	10:	// Nowa operacja rozpoczęta - oczekiwanie na wkręcenie I śruby
		IF bScrewPass THEN
			I_PimSystem.mSetNewMachineState(nPIM_MachineStates._4_OperationInProgress);
			stFastenPIM_Data.i1ScrewPulses := iPassPulses;
			iWorkStep := 15;
		ELSIF NOT fbMotorSensorFilter.Q THEN
			mNewEvent(nEventClass:= nPIM_EventClasses.Error, nEvent:= nHIOS_ErrorList.MotorPulledFromFixWhenLocked);
		END_IF
	
	15:	// wkręcenie 2-giej śruby
		IF bScrewPass THEN
			stFastenPIM_Data.i2ScrewPulses := iPassPulses;
			iWorkStep := 20;
		ELSIF NOT fbMotorSensorFilter.Q THEN
			mNewEvent(nEventClass:= nPIM_EventClasses.Error, nEvent:= nHIOS_ErrorList.MotorPulledFromFixWhenLocked);
		END_IF
	
	20:	// Dwie śruby wkręcone prawidłowo
		I_PimSystem.mSetNewMachineState(nPIM_MachineStates._5_OperationEndedOK);
		iWorkStep := 30;

	30: // Zwolnienie części
		IF I_PimSystem.mSetNewMachineState(nPIM_MachineStates._6_ReturningToBaseState) THEN
			stDigInOuts.bMotorLockValve_Q := FALSE;	
			iWorkStep := 40;
		END_IF
				
	40:	// Operacja zakończona, status zapisany, idź do nowej operacji
		IF NOT fbMotorSensorFilter.Q THEN
			iWorkStep := 1;	
		END_IF	
		
	90:	//  blokowanie stanowiska
		stDigInOuts.bMotorLockValve_Q := TRUE;	
		fbTON_StepTimeout(IN:= FALSE);
		iTypZapytanie := 6;		// Zablokowanie wkrętaka
		iWorkStep := 91;
	
	91:	// Oczekiwanie na zapis statusu, wtedy wystawienie bitu blokowania
		IF I_PimSystem.mSetNewMachineState(nPIM_MachineStates._9_ResetInProgress) OR bServiceReset THEN
			fbTON_StepTimeout(IN:= FALSE);
			bServiceReset := FALSE;
			iWorkStep := 95;
		END_IF

	95:	// Potwierdzenie błędu
		fbTON_StepTimeout(IN:= TRUE, PT := T#2S);
		IF iTypZapytanie = 0 AND NOT bOczekiwanieNaOdpowiedz AND NOT bOdczytOK THEN
			iTypZapytanie := 7;		// Odblokowanie wkrętaka
		END_IF
		IF NOT bWkretakZablokowany THEN	
			stDigInOuts.bMotorLockValve_Q := FALSE;		
			
	
			nError := nHIOS_ErrorList.NoError;
			iWorkStep := 1;	
		END_IF
		IF fbTON_StepTimeout.Q THEN
			mNewEvent(nEventClass:= nPIM_EventClasses.Alarm, nEvent:= nHIOS_ErrorList.ResetTimeout);
		END_IF
		IF iWorkStep <> 95 THEN fbTON_StepTimeout(IN := FALSE); END_IF
	
	ELSE	// Krok domyślny w przypadku błędu w programie
		mNewEvent(nEventClass:= nPIM_EventClasses.Alarm, nEvent:= nHIOS_ErrorList.ProgramConfigError);
END_CASE

ACT_SerialCom();

// Zapis danych PIM	
IF bSqlExtDataSave THEN
	astExtData[1].sName := 'Hios-1Screw[Imp]';
	astExtData[1].sValue := INT_TO_STRING(stFastenPIM_Data.i1ScrewPulses);
	astExtData[2].sName := 'Hios-2Screw[Imp]';
	astExtData[2].sValue := INT_TO_STRING(stFastenPIM_Data.i2ScrewPulses);
	bSqlExtDataSavedOK := I_PimSystem.m_SqlInsertExtendedData(pParameters := ADR(astExtData), uiArraySize := SIZEOF(astExtData));
	bSqlExtDataSave := FALSE;
END_IF

IF GVL_Aircom.stAC_DT_Data.bNew_Shift THEN
	udiNbOfSavedOkStatusesMEM:= udiNbOfSavedOkStatuses;
	udiNbOfSavedNokStatusesMEM := udiNbOfSavedNokStatuses;
	udiNbOfSavedOkStatuses := udiNbOfSavedNokStatuses := 0;
END_IF

ACTION ACT_SerialCom:

IF bReadMachineParams THEN
	IF NOT bSendString AND NOT bOczekiwanieNaOdpowiedz AND NOT bWaitForAllParams THEN	// Start odczytu parametrów
		iTypZapytanie := 1;
		bWaitForAllParams := TRUE;
		iParamsCtr:= 0;
	END_IF
	fbTON_ParamsRead(IN:= bReadMachineParams, PT:= T#2S);
	IF bWaitForAllParams AND iParamsCtr >= 10 THEN			// Gdy wkrętak wysłał wszystkie parametry zakończ odczyt parametrów
		bReadMachineParams := bWaitForAllParams := FALSE;
		fbTON_ParamsRead(IN:=FALSE);
	END_IF
	IF fbTON_ParamsRead.Q THEN		// Parametry nie zostały odczytane
		bWaitForAllParams := bReadMachineParams := FALSE;
		fbTON_ParamsRead(IN:=FALSE);
	END_IF
END_IF

// Komunikacja *************************
fbRTRIG_NewSerialCmd(CLK:= iTypZapytanie <> 0);
bSendString S= fbRTRIG_NewSerialCmd.Q;
IF bSendString THEN
	CASE iTypZapytanie OF
		0:		// Bezczynność
		//	bSendString := FALSE;
		1:		// Zapytanie o parametry
			sSendingString := 'QS$N';
			MEMSET(destAddr := ADR(stScrewDriverParamsAct), fillByte := 0, n := SIZEOF(stScrewDriverParamsAct));
		2:		// Zapytanie o ilosc zalaczen wkretaka
			sSendingString := 'QL$N';
		3:		// Zapytanie o typ wkretaka
			sSendingString := 'QV$N';
		4:		// Reset bledu
			sSendingString := 'R:E$N';
		5:		// Reset licznika śrub do wkręcenia
			sSendingString := 'R:C$N';
		6:		// Zablokowanie wkretaka
			sSendingString := 'Lv:1$N';
		7:		// Odblokowanie wkretaka
			sSendingString := 'Lv:0$N';		
	END_CASE
	
	IF NOT fbSendString.Busy THEN
		sSendStringfb:= sSendingString;
	END_IF
	fbSendString(
		SendString := sSendStringfb,
		TXbuffer := stDigInOuts.stSerialCom.TxBufferEL);
	IF NOT fbSendString.Busy AND (fbSendString.Error = ComError_t.COMERROR_NOERROR) THEN
		MEMMOVE(srcAddr := ADR(asComunicationHistoryOut[1]), destAddr := ADR(asComunicationHistoryOut[2]),n:= 9* SIZEOF(asComunicationHistoryOut[1]));
		asComunicationHistoryOut[1]:= sSendStringfb;
		bSendString := FALSE;
		bOczekiwanieNaOdpowiedz:=TRUE;	
	ELSIF NOT fbSendString.Busy AND (fbSendString.Error <> ComError_t.COMERROR_NOERROR) THEN
		bSendString := FALSE;
		iTypZapytanie := 0;
		fbRTRIG_NewSerialCmd(CLK := FALSE);
		bOczekiwanieNaOdpowiedz:=FALSE;
		iComSendError := fbSendString.Error;	
	END_IF
END_IF 

fbRecvString(Prefix :='',
		Suffix := '$N',
		Timeout := T#1S,
		Reset := ,
		StringReceived =>,
		Busy =>,
		RXbuffer := stDigInOuts.stSerialCom.RxBufferEL,
		ReceivedString := sRcvString);

// Sprawdzenie poprawności komunikacji oraz odebranych danych
fbTON_Timer_Comm(IN := bSendString OR bOczekiwanieNaOdpowiedz, PT:= T#2S);

IF fbTON_Timer_Comm.Q THEN
	bQBladKomunikacji := TRUE;
	bOczekiwanieNaOdpowiedz := FALSE;
	bSendString:= FALSE;
	bOdczytOK := FALSE;
	fbRTRIG_NewSerialCmd(CLK := FALSE);
	iTypZapytanie := 0;
END_IF
// Dekodowanie odebranych informacji
bTorqueUp := bScrewFail := bScrewPass := FALSE;
bOdczytOK := FALSE;
IF fbRecvString.StringReceived THEN
	sRcvString := DELETE(STR:= sRcvString, LEN:=1, POS:= LEN(sRcvString));
	MEMMOVE(srcAddr := ADR(asComunicationHistoryIn[1]), destAddr := ADR(asComunicationHistoryIn[2]),n:= 9* SIZEOF(asComunicationHistoryIn[1]));
	asComunicationHistoryIn[1]:= sRcvString;
	bQBladKomunikacji := FALSE;
	bOczekiwanieNaOdpowiedz := FALSE;
	bOdczytOK := TRUE;
	iTypZapytanie := 0;
	// Wyłuskanie parametrow
	// Actual values	
	IF FIND(sRcvString, 'Lv:') > 0 THEN			// Określenie czy wkretak jest zablokowany
		sStringToRead := DELETE(STR:= sRcvString, LEN := 3, POS :=1);
		bWkretakZablokowany := STRING_TO_INT(sStringToRead) > 0;
	ELSIF FIND(sRcvString, 'AL:') > 0 THEN		// Licznik uruchomień
		sStringToRead := DELETE(STR:= sRcvString, LEN := 3, POS :=1);
		diStartsUpCtr := STRING_TO_DINT(sStringToRead);	
	ELSIF FIND(sRcvString, 'L:') > 0 THEN			// Określenie czy wkretak jest wlaczony
		sStringToRead := DELETE(STR:= sRcvString, LEN := 2, POS :=1);
		IF STRING_TO_INT(sStringToRead) > 0 THEN
			bWkretakWlaczony := TRUE;
			diStartsUpCtr := diStartsUpCtr +1;
		ELSE
			bWkretakWlaczony := FALSE;
		END_IF
	ELSIF FIND(sRcvString, 'Pulse:') > 0 THEN			// Aktualny licznik impulsow
		sStringToRead := DELETE(STR:= sRcvString, LEN := 6, POS :=1);
		iActPulses:= STRING_TO_INT(sStringToRead);
	ELSIF FIND(sRcvString, 'PASS') > 0 THEN			// Śruba wkręcona prawidlowo
		bScrewPass := TRUE;
	ELSIF FIND(sRcvString, 'FAIL') > 0 THEN			// Śruba wkręcona błędnie
		bScrewFail := TRUE;
	ELSIF FIND(sRcvString, 'E:  ,') > 0 THEN		// Licznik impulsow - bledna sruba
		sStringToRead := DELETE(STR:= sRcvString, LEN := 5, POS :=1);
		iFailPulses:= STRING_TO_INT(sStringToRead);
	ELSIF FIND(sRcvString, 'D:') > 0 THEN		// Licznik impulsow - dobra sruba
		sStringToRead := DELETE(STR:= sRcvString, LEN := 7, POS :=1);
		iPassPulses:= STRING_TO_INT(sStringToRead);
	ELSIF FIND(sRcvString, 'T') > 0 THEN		// Osiagnieto moment
		bTorqueUp:= TRUE;
	// Parameters
	ELSIF FIND(sRcvString, 'AR:') > 0 THEN			// Maksymalna liczba impulsow
		sStringToRead := DELETE(STR:= sRcvString, LEN := 3, POS :=1);
		stScrewDriverParamsAct.iSystemConstAR := STRING_TO_INT(sStringToRead);
		iParamsCtr := iParamsCtr + 1;
	ELSIF FIND(sRcvString, 'An:') > 0 THEN			// Liczba śrub do wkrecenia
		sStringToRead := DELETE(STR:= sRcvString, LEN := 3, POS :=1);
		stScrewDriverParamsAct.iScrewsToFastenAn := STRING_TO_INT(sStringToRead);
		iParamsCtr := iParamsCtr + 1;
	ELSIF FIND(sRcvString, 'Ac:') > 0 THEN			// Minimalna liczba impulsow
		sStringToRead := DELETE(STR:= sRcvString, LEN := 3, POS :=1);
		stScrewDriverParamsAct.iMinPulseAc := STRING_TO_INT(sStringToRead);
		iParamsCtr := iParamsCtr + 1;
	ELSIF FIND(sRcvString, 'AC:') > 0 THEN			// Maksymalna liczba impulsow
		sStringToRead := DELETE(STR:= sRcvString, LEN := 3, POS :=1);
		stScrewDriverParamsAct.iMaxPulseAC := STRING_TO_INT(sStringToRead);
		iParamsCtr := iParamsCtr + 1;
	ELSIF FIND(sRcvString, 'At:') > 0 THEN			// Work reset time
		sStringToRead := DELETE(STR:= sRcvString, LEN := 3, POS :=1);
		stScrewDriverParamsAct.iBuzzerScrewsDoneTimeAt := STRING_TO_INT(sStringToRead);
		iParamsCtr := iParamsCtr + 1;
	ELSIF FIND(sRcvString, 'Ar:') > 0 THEN			// Count time for reverse operation
		sStringToRead := DELETE(STR:= sRcvString, LEN := 3, POS :=1);
		stScrewDriverParamsAct.iCntTimeForReverseOperationAr := STRING_TO_INT(sStringToRead);
		iParamsCtr := iParamsCtr + 1;
	ELSIF FIND(sRcvString, 'Ad:') > 0 THEN			// System setting
		sStringToRead := DELETE(STR:= sRcvString, LEN := 3, POS :=1);
		stScrewDriverParamsAct.iSystemSettingAd := STRING_TO_INT(sStringToRead);
		iParamsCtr := iParamsCtr + 1;
	ELSIF FIND(sRcvString, 'AU:') > 0 THEN			// Error detection setting
		sStringToRead := DELETE(STR:= sRcvString, LEN := 3, POS :=1);
		stScrewDriverParamsAct.iErrorTypesDetectionAU := STRING_TO_INT(sStringToRead);	
		iParamsCtr := iParamsCtr + 1;
	ELSIF FIND(sRcvString, 'Ao:') > 0 THEN			// Operation panel button enable
		sStringToRead := DELETE(STR:= sRcvString, LEN := 3, POS :=1);
		stScrewDriverParamsAct.iOperPanelButtonsEnableAo := STRING_TO_INT(sStringToRead);
		iParamsCtr := iParamsCtr + 1;	
	ELSIF FIND(sRcvString, 'AG:') > 0 THEN			// Inactive time after PASS / FAIL
		sStringToRead := DELETE(STR:= sRcvString, LEN := 3, POS :=1);
		stScrewDriverParamsAct.iInactiveTimeAfterP_FAG := STRING_TO_INT(sStringToRead);	
		iParamsCtr := iParamsCtr + 1;
	ELSIF FIND(sRcvString, 'R') > 0 THEN		// Zmieniono liczbę srub do wkręcenia
		bScrewsQuantityCHanged:= TRUE;
	ELSIF FIND(sRcvString, 'Over') > 0 THEN		// Konieczny przeglad - milion śrub wkręconych)
		bMaintenanceRequest:= TRUE;
		nError := nHIOS_ErrorList.OverMilion_ResetReq;
	ELSIF FIND(sRcvString, 'CE:') > 0 THEN		// Kod Bledu
		sErrorString := DELETE(STR:= sRcvString, LEN := 3, POS :=1);
	ELSIF FIND(sRcvString, 'Ver') > 0 THEN		// Wersja urzadzenia
		sVersionType := sRcvString;
	END_IF
	
END_IF
END_ACTION

METHOD FB_init : BOOL
VAR_INPUT
	bInitRetains : BOOL; // if TRUE, the retain variables are initialized (warm start / cold start)
	bInCopyCode : BOOL;  // if TRUE, the instance afterwards gets moved into the copy code (online change)
	I_Pim	: I_PIM;		// Interfejs do bloku PIM
END_VAR
I_PimSystem := I_Pim;
END_METHOD

(* Metoda TRUE kiedy dane wyjściowe są ok, jeśli nie FALSE (jeśli not bBusy i FALSE to błąd odczytu) *)
METHOD mGetParamsData : BOOL
VAR_INPUT
	bTestParams:	BOOL;	// Jeśli TRUE metoda okresla czy ma dostęp do parametrów, jeśli tak zwraca TRUE, jeśli nie FALSE
END_VAR
VAR_OUTPUT
	bBusy	: BOOL;										//	Maszyna odświeża dane
	pMachineParametersStruct	: POINTER TO BYTE;		// 	Wskaźnik do parametrów pracy maszyny
	uiMachineParametersSize	: UINT;						// 	Rozmiar struktury parametrów pracy maszyny [bajty]
	wActualCRC16SumInMachine	: WORD;					//	Aktualna suma CRC16 obliczona z parametrów
END_VAR
IF bTestParams THEN
	mGetParamsData := FALSE;
ELSE
	pMachineParametersStruct := 0;
	uiMachineParametersSize := 0;
	wActualCRC16SumInMachine := F_DATA_TO_CRC16_CCITT(pData := pMachineParametersStruct, cbData := uiMachineParametersSize, crc := 16#0000);
	bBusy := FALSE;
	mGetParamsData := TRUE;
END_IF
END_METHOD

METHOD INTERNAL mNewEvent : BOOL
VAR_INPUT
	nEventClass:nPIM_EventClasses;
	nEvent: nHIOS_ErrorList;
END_VAR
IF nEventClass = nPIM_EventClasses.AlarmAutoConfirm OR nEventClass = nPIM_EventClasses.Message THEN		// Alarm nieblokadowy
	I_PimSystem.mSetNewMachineState(nPIM_MachineStates._0_Initialization);
	iWorkStep := 95;
ELSE
	I_PimSystem.mSetNewMachineState(nPIM_MachineStates._7_ErrorOccurr);
	I_PimSystem.mNewEvent(iEventId := nEvent, nEventType := nEventClass, tMessageTime := T#0S);
	iWorkStep := 90;
END_IF
nError := nEvent;
END_METHOD

END_FUNCTION_BLOCK

// ProdLineMachines/S13_FrontFanPress/fbFrontFanPress
FUNCTION_BLOCK fbFrontFanPress IMPLEMENTS I_StationMachine
VAR_IN_OUT
	stInOuts: stFrontFanPress_InOuts;
END_VAR
VAR_INPUT
	tDeltaDwuStart:TIME:= T#200MS;
END_VAR
VAR_OUTPUT
	bStabilizerValve_Q:BOOL;	// Sygnał do układu stabilizującego części przed wprasowaniem - 1 - stabilizacja części
	bPressValve_Q:BOOL;	// Sygnał do zaworu sterującego prasą - 1 - wprasowywanie
	nError:nFrontFanPress_ErrorCodes;
END_VAR
VAR
	I_PimSystem			: I_PIM;
	fb2Start: fb2HandStartBasic;
	iWorkStep: INT;
	udiOperationsOK_Qty: UDINT;
	iTmpConv: INT;
	fbTON_StabilizerWorkPos: TON;
	fbTON_StepTimeout: TON;
	tLastNoNcContactsDiffTime: TIME;
	bServiceReset: BOOL;
END_VAR

fb2Start(stInOutsData:= stInOuts.st2HandStartIO, tDeltaDwuStart := T#250MS);

//  Błędy monitorowane stale (bezpieczeństwo)
IF NOT stInOuts.st2HandStartIO.bEmergButton_NC AND nError <> nFrontFanPress_ErrorCodes.SafetySystemNotArmed THEN
	stInOuts.bPressValve_Q := stInOuts.bStabilizerValve_Q := FALSE;
	mNewEvent(nEvent:=nFrontFanPress_ErrorCodes.SafetySystemNotArmed , nEventClass := nPIM_EventClasses.Error);
END_IF

CASE iWorkStep OF 
	0:	// Inicjalizacja
		I_PimSystem.mSetNewMachineState(nPIM_MachineStates._0_Initialization);
		iWorkStep := 1;
		
	1:	// Init
		I_PimSystem.mSetNewMachineState(nPIM_MachineStates._0_Standby_NotReady);
		stInOuts.bPressValve_Q := stInOuts.bStabilizerValve_Q := FALSE;
		iWorkStep := 5;
	
	5:	// Krok spoczynkowy - oczekiwanie na nową operację
		I_PimSystem.mSetNewMachineState(nPIM_MachineStates._2_ReadyForNewOperation);
		IF fb2Start.bStartSig THEN
			IF stInOuts.bPressHomePos AND_THEN I_PimSystem.mSetNewMachineState(nPIM_MachineStates._3_NewOperationStarted) THEN 
				iWorkStep := 10;
				fbTON_StabilizerWorkPos(IN:= FALSE);
				fbTON_StepTimeout(IN:= FALSE);				
			ELSIF NOT stInOuts.bPressHomePos THEN
				I_PimSystem.mNewServiceMessage(sMessage := 'Press is not in home possition',tMessageTime := T#5S);	
			ELSIF NOT I_PimSystem.mSetNewMachineState(nPIM_MachineStates._3_NewOperationStarted) THEN 
				I_PimSystem.mNewServiceMessage(sMessage := 'No Work permition from PIM system',tMessageTime := T#5S);	
			END_IF
		END_IF
		
	10:	// Nowa operacja rozpoczęta - stabilizacja części
		IF fb2Start.bStartSig THEN
			stInOuts.bStabilizerValve_Q := TRUE;
			fbTON_StepTimeout(IN:= TRUE, PT:= T#1S);
			fbTON_StabilizerWorkPos(IN:= NOT stInOuts.bStabilizerHomePos, PT:= T#300MS);
			IF fbTON_StabilizerWorkPos.Q THEN	// Jest ruch siłownika
				iWorkStep := 15;
			ELSIF fbTON_StepTimeout.Q THEN
				I_PimSystem.mNewServiceMessage(sMessage := 'No stabilizer reaction',tMessageTime := T#5S);	
				stInOuts.bStabilizerValve_Q := FALSE;
				mNewEvent(nEventClass:= nPIM_EventClasses.Alarm, nEvent:= nFrontFanPress_ErrorCodes.StabilizingTimeout);
			END_IF	
		ELSE
			stInOuts.bStabilizerValve_Q := FALSE;
			iWorkStep := 5;
		END_IF	
		IF iWorkStep <> 10 THEN fbTON_StepTimeout(IN:= FALSE); fbTON_StabilizerWorkPos(IN:= FALSE); END_IF
	
	15:	// Oczekiwanie na osiągnięcie pozycji roboczej
		IF fb2Start.bStartSig THEN
			fbTON_StepTimeout(IN:= TRUE, PT:= T#1S);
			stInOuts.bPressValve_Q := TRUE;
			IF stInOuts.bPressWorkPos THEN	// Pozycja docelowa osiągnięta
				I_PimSystem.mSetNewMachineState(nPIM_MachineStates._4_OperationInProgress);
				iWorkStep := 20;
			ELSIF fbTON_StepTimeout.Q THEN
				stInOuts.bPressValve_Q := stInOuts.bStabilizerValve_Q := FALSE;
				mNewEvent(nEventClass:= nPIM_EventClasses.Error, nEvent:= nFrontFanPress_ErrorCodes.WorkPosAchieveTimeout);
			END_IF	
		ELSE
			stInOuts.bPressValve_Q := stInOuts.bStabilizerValve_Q := FALSE;
			mNewEvent(nEventClass:= nPIM_EventClasses.Alarm, nEvent:= nFrontFanPress_ErrorCodes.OperInteruptedBeforeWorkPos);
		END_IF	
		IF iWorkStep <> 15 THEN fbTON_StepTimeout(IN:= FALSE); END_IF
			
	20:	// Prasa w pozycji roboczej - oczekiwanie przez zadany czas
		fbTON_StepTimeout(IN:= TRUE, PT := T#500MS);
		IF NOT stInOuts.bPressWorkPos THEN
			mNewEvent(nEventClass:= nPIM_EventClasses.Error, nEvent:= nFrontFanPress_ErrorCodes.WorkPosLost);
		ELSIF fbTON_StepTimeout.Q THEN
			udiOperationsOK_Qty := udiOperationsOK_Qty +1;
			I_PimSystem.mSetNewMachineState(nPIM_MachineStates._5_OperationEndedOK);
			iWorkStep := 25;
		END_IF
		IF iWorkStep <> 20 THEN	fbTON_StepTimeout(IN:= FALSE); END_IF
		
	25:	// Cofnięcie prasy
		fbTON_StepTimeout(IN:= TRUE, PT := T#1S);
		stInOuts.bPressValve_Q := FALSE;
		IF stInOuts.bPressHomePos THEN
			iWorkStep := 30;	
		ELSIF fbTON_StepTimeout.Q THEN
			mNewEvent(nEventClass:= nPIM_EventClasses.Alarm, nEvent:= nFrontFanPress_ErrorCodes.HomePosAchieveTimeout);
		END_IF
		IF iWorkStep <> 25 THEN	fbTON_StepTimeout(IN:= FALSE); END_IF

	
	30:	// Zakończenie operacji		 
		IF I_PimSystem.mSetNewMachineState(nPIM_MachineStates._6_ReturningToBaseState) THEN
			iWorkStep := 31;
		END_IF
		
	31:	// Cofnięcie stabilizatora
		fbTON_StepTimeout(IN:= TRUE, PT := T#1S);
		stInOuts.bStabilizerValve_Q := FALSE;
		IF stInOuts.bStabilizerHomePos THEN
			iWorkStep := 35;
		ELSIF fbTON_StepTimeout.Q THEN
			mNewEvent(nEventClass:= nPIM_EventClasses.Error, nEvent:= nFrontFanPress_ErrorCodes.StabilizerReturnTimeout);		// Błąd powrotu do pozycji bazowej
		END_IF
		IF iWorkStep <> 31 THEN	fbTON_StepTimeout(IN:= FALSE); END_IF
				
	35:	// Czekanie na zwolnienie dwustartu i podniesienie uchwytu (wyciągnięcie części)
		IF NOT fb2Start.bStartSig THEN
			iWorkStep := 5;
		END_IF
		
	90:	// Zapis statusu NOK i blokowanie stanowiska
		stInOuts.bPressValve_Q := stInOuts.bPressWorkPos;
		stInOuts.bStabilizerValve_Q := NOT stInOuts.bStabilizerHomePos;
		I_PimSystem.mSetNewMachineState(nPIM_MachineStates._8_WaitForReset);
		iWorkStep := 91;
		
	91:	// Oczekiwanie na potwierdzenie
		IF I_PimSystem.mSetNewMachineState(nPIM_MachineStates._9_ResetInProgress) OR bServiceReset THEN
			bServiceReset := FALSE;
			fbTON_StepTimeout(IN:= FALSE);
			iWorkStep := 95;
		END_IF
		
	95:	// Potwierdzenie błedu
		IF NOT stInOuts.st2HandStartIO.bEmergButton_NC THEN
			mNewEvent(nEventClass:= nPIM_EventClasses.Error, nEvent:= nFrontFanPress_ErrorCodes.SafetySystemNotArmed);
		ELSE
			stInOuts.bPressValve_Q := FALSE;
			stInOuts.bStabilizerValve_Q R= stInOuts.bPressHomePos;
			IF stInOuts.bPressHomePos AND stInOuts.bStabilizerHomePos AND stInOuts.st2HandStartIO.bEmergButton_NC AND fbTON_StepTimeout.ET > T#200MS THEN
				nError := nFrontFanPress_ErrorCodes.NoError;
				I_PimSystem.mSetNewMachineState(nPIM_MachineStates._0_Standby_NotReady);
				iWorkStep := 0 ;	// Powrót do kroku inicjalizacyjnego lub wskazanego w algorytmie
			END_IF
		END_IF
		fbTON_StepTimeout(IN:= TRUE, PT := T#3S);
		IF fbTON_StepTimeout.Q THEN
			mNewEvent(nEventClass:= nPIM_EventClasses.Error, nEvent:= nFrontFanPress_ErrorCodes.ResetTimeout);
		END_IF

	ELSE	// Krok domyślny w przypadku błędu w programie
		mNewEvent(nEventClass:= nPIM_EventClasses.Error, nEvent:= nFrontFanPress_ErrorCodes.ProgramConfigError);		
END_CASE

stInOuts.bPressValve_Q R= stInOuts.bStabilizerValve_Q R= NOT stInOuts.st2HandStartIO.bEmergButton_NC;

METHOD FB_init : BOOL
VAR_INPUT
	bInitRetains : BOOL; // if TRUE, the retain variables are initialized (warm start / cold start)
	bInCopyCode : BOOL;  // if TRUE, the instance afterwards gets moved into the copy code (online change)
	I_Pim	: I_PIM;		// Interfejs do bloku PIM
END_VAR
I_PimSystem := I_Pim;
END_METHOD

(* Metoda TRUE kiedy dane wyjściowe są ok, jeśli nie FALSE (jeśli not bBusy i FALSE to błąd odczytu) *)
METHOD mGetParamsData : BOOL
VAR_INPUT
	bTestParams:	BOOL;	// Jeśli TRUE metoda okresla czy ma dostęp do parametrów, jeśli tak zwraca TRUE, jeśli nie FALSE
END_VAR
VAR_OUTPUT
	bBusy	: BOOL;										//	Maszyna odświeża dane
	pMachineParametersStruct	: POINTER TO BYTE;		// 	Wskaźnik do parametrów pracy maszyny
	uiMachineParametersSize	: UINT;						// 	Rozmiar struktury parametrów pracy maszyny [bajty]
	wActualCRC16SumInMachine	: WORD;					//	Aktualna suma CRC16 obliczona z parametrów
END_VAR
IF bTestParams THEN
	mGetParamsData := FALSE;
ELSE
	pMachineParametersStruct := 0;
	uiMachineParametersSize := 0;
	wActualCRC16SumInMachine := F_DATA_TO_CRC16_CCITT(pData := pMachineParametersStruct, cbData := uiMachineParametersSize, crc := 16#0000);
	bBusy := FALSE;
	mGetParamsData := TRUE;
END_IF
END_METHOD

METHOD INTERNAL mNewEvent : BOOL
VAR_INPUT
	nEventClass:nPIM_EventClasses;
	nEvent: nFrontFanPress_ErrorCodes;
END_VAR
IF nEventClass = nPIM_EventClasses.AlarmAutoConfirm OR nEventClass = nPIM_EventClasses.Message THEN		// Alarm nieblokadowy
	I_PimSystem.mSetNewMachineState(nPIM_MachineStates._0_Initialization);
	iWorkStep := 95;
ELSE
	I_PimSystem.mSetNewMachineState(nPIM_MachineStates._7_ErrorOccurr);
	I_PimSystem.mNewEvent(iEventId := nEvent, nEventType := nEventClass, tMessageTime := T#0S);
	iWorkStep := 90;
END_IF
nError := nEvent;
END_METHOD

END_FUNCTION_BLOCK

// ProdLineMachines/S18_ManometerCalib/fbManometerCalibration
FUNCTION_BLOCK fbManometerCalibration IMPLEMENTS I_StationMachine
VAR_IN_OUT
	stInOuts: stManometerCalibration_InOuts;
END_VAR
VAR_INPUT
	stTestParams:stManometerCalibration_TestData;
	stHwSettings:stMeasurementScalingData;
	bCompressorSensorInvert: BOOL:= FALSE;
END_VAR
VAR_OUTPUT
	nError:nManometerCalibration_ErrorCodes;
END_VAR
VAR
	I_PimSystem			: I_PIM;
	fb2Start: fb2HandStartBasic;
	fbPressureMeasure:fbAnalogMeasurement;
	fbFilterCompressorSensor: fbBinaryFilter;
	fbformat: FB_FormatString;
	udiOperationsOK_Qty: UDINT;
	iWorkStep: INT;
	fbTON_StepTimeout: TON;					// Timer timeoutu kroku algorytmu
	rPressureValue: REAL;					// Wartość pomiaru ciśnienia ustawczego
	fbTON_PressureOutOfRangeErr: TON;		// Timer przekroczenia zakresu dopuszczalnego ciśnienia skalowania
	udiNbOfSavedOkStatuses,	udiNbOfSavedNokStatuses, udiNbOfSavedOkStatusesMEM, udiNbOfSavedNokStatusesMEM: UDINT;	// Liczniki zapusanych statusów PIM
	bServiceReset: BOOL;
END_VAR

// Pomiar ciśnienia
fbPressureMeasure( rIn:= INT_TO_REAL(stInOuts.iPressure), 
	bExtError:= stInOuts.bPressureSensorError, 
	stMeasureScalingData:= stHwSettings, 
	tStalaCzasowa:= T#200MS, 
	rOutFiltered=> rPressureValue);

fb2Start(stInOutsData:= stInOuts.st2HandStartIO, tDeltaDwuStart := T#350MS);
	
//  Błędy monitorowane stale (bezpieczeństwo)
IF NOT stInOuts.st2HandStartIO.bEmergButton_NC AND nError <> nManometerCalibration_ErrorCodes.SafetySystemNotArmed THEN
	stInOuts.bNozzlePusherValve_Q := stInOuts.bTargetAirValve_Q := FALSE;
	stInOuts.bTestFrameCloseValve_Q := stInOuts.bTestFrameOpenValve_Q := FALSE;
	mNewEvent(nEvent:=nManometerCalibration_ErrorCodes.SafetySystemNotArmed , nEventClass := nPIM_EventClasses.Error);
END_IF

// Dopasowanie poziomów
fbFilterCompressorSensor(IN := stInOuts.bCompressorSensor XOR bCompressorSensorInvert, tON:= T#100MS, tOFF := T#100MS);

CASE iWorkStep OF 
	0:	// Inicjalizacja
		I_PimSystem.mSetNewMachineState(nPIM_MachineStates._0_Initialization);
		stInOuts.bNozzlePusherValve_Q := stInOuts.bNozzlePusherWorkPos;
		stInOuts.bTargetAirValve_Q := FALSE;
		stInOuts.bTestFrameCloseValve_Q := stInOuts.bTestFrameHomePos AND NOT stInOuts.bTestFrameWorkPos;
		stInOuts.bTestFrameOpenValve_Q := stInOuts.bTestFrameWorkPos AND NOT stInOuts.bTestFrameHomePos;
		fbTON_StepTimeout(IN:= FALSE);
		iWorkStep := 1;
		
	1:	// Init
		I_PimSystem.mSetNewMachineState(nPIM_MachineStates._0_Standby_NotReady);
		fbTON_StepTimeout(IN:= TRUE, PT:= T#2S);
		IF stInOuts.bTestFrameHomePos AND stInOuts.bNozzlePusherHomePos THEN
			iWorkStep := 5;
			stInOuts.bTestFrameCloseValve_Q := TRUE; 
			stInOuts.bTestFrameOpenValve_Q := stInOuts.bNozzlePusherValve_Q := stInOuts.bTargetAirValve_Q := FALSE;
		ELSIF fbTON_StepTimeout.Q THEN
			mNewEvent(nEventClass:= nPIM_EventClasses.Alarm, nEvent:= nManometerCalibration_ErrorCodes.StationResetRequired);
		END_IF
		IF iWorkStep <> 1 THEN fbTON_StepTimeout(IN:= FALSE); END_IF
	
	5:	// Krok spoczynkowy - oczekiwanie na nową operację
		I_PimSystem.mSetNewMachineState(nPIM_MachineStates._2_ReadyForNewOperation);
		IF fb2Start.bStartSig THEN
			IF fbFilterCompressorSensor.Q AND_THEN I_PimSystem.mSetNewMachineState(nPIM_MachineStates._3_NewOperationStarted) THEN 
				iWorkStep := 10;
				fbTON_StepTimeout(IN:= FALSE);
			ELSIF NOT fbFilterCompressorSensor.Q THEN
				I_PimSystem.mNewServiceMessage(sMessage := 'No compressor detected',tMessageTime := T#5S);	
			ELSIF NOT I_PimSystem.mSetNewMachineState(nPIM_MachineStates._3_NewOperationStarted) THEN
				I_PimSystem.mNewServiceMessage(sMessage := 'No Work permition from PIM system',tMessageTime := T#5S);	
			END_IF
		END_IF
		
	10:	// Nowa operacja rozpoczęta - sprawdzenie ciśnienia wzorcowania
		IF fb2Start.bStartSig THEN
			IF stTestParams.bPressureCheckingEN AND (ABS(rPressureValue- stTestParams.rSettingPressure) > stTestParams.rSettingPressureDeviation) THEN
				mNewEvent(nEventClass:= nPIM_EventClasses.Alarm, nEvent:= nManometerCalibration_ErrorCodes.PressureOutOfRange);		
				fbformat(sFormat:= 'Calibration pressure outside the desired range- %.2f[bar] (desired %.2f +- %.2f[bar])',
						arg1 := F_REAL(rPressureValue), arg2:= F_REAL(stTestParams.rSettingPressure), arg3 := F_REAL(stTestParams.rSettingPressureDeviation));
				I_PimSystem.mNewServiceMessage(sMessage := fbformat.sOut,tMessageTime := T#5S);	
			ELSE
				iWorkStep := 15;
			END_IF	
		ELSE
			iWorkStep := 5;
		END_IF	
	
	15:	// Wysunięcie ramienia pomiarowego - sprawdzenie reakcji
		IF fb2Start.bStartSig THEN
			fbTON_StepTimeout(IN:= TRUE, PT:= T#1S);
			stInOuts.bTestFrameCloseValve_Q := FALSE;
			stInOuts.bTestFrameOpenValve_Q := TRUE;
			IF NOT stInOuts.bTestFrameHomePos THEN	// Ramię ruszyło
				iWorkStep := 20;
			ELSIF fbTON_StepTimeout.Q THEN
				I_PimSystem.mNewServiceMessage(sMessage := 'No reaction to piston open signal- low pressure or valve malfunction',tMessageTime := T#5S);	
				stInOuts.bTestFrameCloseValve_Q := stInOuts.bTestFrameOpenValve_Q := FALSE;
				mNewEvent(nEventClass:= nPIM_EventClasses.Error, nEvent:= nManometerCalibration_ErrorCodes.NoMachineReactionOnStartSig);
			END_IF
		ELSE
			stInOuts.bTestFrameCloseValve_Q := TRUE;
			stInOuts.bTestFrameOpenValve_Q := FALSE;
			iWorkStep := 5;
		END_IF	
		IF iWorkStep <> 15 THEN fbTON_StepTimeout(IN:= FALSE); END_IF	
			
	20:	// Wysunięcie ramienia testowego - oczekiwanie na pozycję docelową
		IF fb2Start.bStartSig THEN
			fbTON_StepTimeout(IN:= TRUE, PT:= T#2S);
			stInOuts.bTestFrameCloseValve_Q := FALSE;
			stInOuts.bTestFrameOpenValve_Q := TRUE;
			IF stInOuts.bTestFrameWorkPos THEN	// Ramię w pozycji docelowej
				iWorkStep := 25;
			ELSIF fbTON_StepTimeout.Q THEN
				stInOuts.bTestFrameCloseValve_Q := stInOuts.bTestFrameOpenValve_Q := FALSE;
				I_PimSystem.mNewServiceMessage(sMessage := 'Frame work position not achieved - lock of piston or invalid set end sensor',tMessageTime := T#5S);	
				mNewEvent(nEventClass:= nPIM_EventClasses.Error, nEvent:= nManometerCalibration_ErrorCodes.WorkPosAchieveTimeout);
			END_IF
		ELSE
			stInOuts.bTestFrameCloseValve_Q := TRUE;
			stInOuts.bTestFrameOpenValve_Q := FALSE;
			mNewEvent(nEventClass:= nPIM_EventClasses.Alarm, nEvent:= nManometerCalibration_ErrorCodes.OperInteruptedBeforeWorkPos);
		END_IF	
		IF iWorkStep <> 20 THEN fbTON_StepTimeout(IN:= FALSE); END_IF	

	25: // Wysunięcie/podłączenie dyszy	
		IF fb2Start.bStartSig THEN
			fbTON_StepTimeout(IN:= TRUE, PT:= T#1S);
			stInOuts.bNozzlePusherValve_Q := TRUE;
			IF stInOuts.bNozzlePusherWorkPos THEN
				iWorkStep := 30;
			ELSIF fbTON_StepTimeout.Q THEN
				stInOuts.bNozzlePusherValve_Q := FALSE;
				I_PimSystem.mNewServiceMessage(sMessage := 'Nozzle work position not achieved - lock of piston or invalid set end sensor',tMessageTime := T#5S);	
				mNewEvent(nEventClass:= nPIM_EventClasses.Error, nEvent:= nManometerCalibration_ErrorCodes.WorkPosAchieveTimeout);
			END_IF	
		ELSE
			stInOuts.bNozzlePusherValve_Q := FALSE;
			mNewEvent(nEventClass:= nPIM_EventClasses.Error, nEvent:= nManometerCalibration_ErrorCodes.OperInteruptedBeforeWorkPos);
		END_IF	
		IF iWorkStep <> 25 THEN fbTON_StepTimeout(IN:= FALSE); END_IF
			
	30:	// Układ w pozycji testowej - oczekiwanie na uszczelnienie i podanie ciśnienia 
		fbTON_StepTimeout(IN:= TRUE, PT:= T#400MS);
		stInOuts.bTargetAirValve_Q S= fbTON_StepTimeout.ET > T#300MS;
		IF fbTON_StepTimeout.Q AND NOT fb2Start.bStartSig THEN
			I_PimSystem.mSetNewMachineState(nPIM_MachineStates._4_OperationInProgress);
			iWorkStep := 35;
		END_IF
		IF iWorkStep <> 30 THEN fbTON_StepTimeout(IN:= FALSE); END_IF

	35:	// Naklejanie etykiety
		fbTON_StepTimeout(IN:= NOT stInOuts.bNozzlePusherWorkPos, PT:= T#1M);
		stInOuts.bTargetAirValve_Q := TRUE;	
		IF fb2Start.bStartSig THEN
			udiOperationsOK_Qty := udiOperationsOK_Qty +1;
			stInOuts.bTargetAirValve_Q := FALSE;
			I_PimSystem.mSetNewMachineState(nPIM_MachineStates._5_OperationEndedOK);
			iWorkStep := 40;
		END_IF
		IF stTestParams.bPressureCheckingEN THEN
			fbTON_PressureOutOfRangeErr(IN:= ABS(rPressureValue- stTestParams.rSettingPressure) > stTestParams.rSettingPressureDeviation, PT:= T#500MS);
			IF fbTON_PressureOutOfRangeErr.Q THEN
				mNewEvent(nEventClass:= nPIM_EventClasses.Error, nEvent:= nManometerCalibration_ErrorCodes.PressureOutOfRange);
				fbformat(sFormat:= 'Calibration pressure outside the desired range- %.2f[bar] (desired %.2f +- %.2f[bar])',
						arg1 := F_REAL(rPressureValue), arg2:= F_REAL(stTestParams.rSettingPressure), arg3 := F_REAL(stTestParams.rSettingPressureDeviation));
				I_PimSystem.mNewServiceMessage(sMessage := fbformat.sOut,tMessageTime := T#5S);	
			END_IF
		ELSIF fbTON_StepTimeout.Q THEN
			mNewEvent(nEventClass:= nPIM_EventClasses.Error, nEvent:= nManometerCalibration_ErrorCodes.OprationTooLong);
		ELSE
			fbTON_PressureOutOfRangeErr(IN:= FALSE);
		END_IF
		IF iWorkStep <> 35 THEN	fbTON_StepTimeout(IN:= FALSE); END_IF
		
	
	40:	// Powrót do stanu początkowego		 
		IF I_PimSystem.mSetNewMachineState(nPIM_MachineStates._6_ReturningToBaseState) THEN
			iWorkStep := 45;
		END_IF
		
	45:	// Cofnięcie siłowników
		fbTON_StepTimeout(IN:= TRUE, PT := T#4S);
		stInOuts.bNozzlePusherValve_Q := fbTON_StepTimeout.ET < T#200MS;
		IF stInOuts.bNozzlePusherHomePos THEN
			stInOuts.bTestFrameCloseValve_Q := TRUE;
			stInOuts.bTestFrameOpenValve_Q := FALSE;
			IF stInOuts.bTestFrameHomePos THEN
				iWorkStep := 50;	
			END_IF
		ELSIF fbTON_StepTimeout.Q THEN
			mNewEvent(nEventClass:= nPIM_EventClasses.Alarm, nEvent:= nManometerCalibration_ErrorCodes.HomePosAchieveTimeout);
		END_IF
		IF iWorkStep <> 45 THEN	fbTON_StepTimeout(IN:= FALSE); END_IF
	
				
	50:	// Czekanie na zwolnienie dwustartu i podniesienie uchwytu (wyciągnięcie części)
		IF NOT fb2Start.bStartSig AND NOT fbFilterCompressorSensor.Q THEN
			iWorkStep := 5;
		END_IF
		
	90:	// Zapis statusu NOK i blokowanie stanowiska
		stInOuts.bNozzlePusherValve_Q := stInOuts.bNozzlePusherWorkPos;
		stInOuts.bTargetAirValve_Q := FALSE;
		stInOuts.bTestFrameCloseValve_Q := stInOuts.bTestFrameHomePos AND NOT stInOuts.bTestFrameWorkPos;
		stInOuts.bTestFrameOpenValve_Q := stInOuts.bTestFrameWorkPos AND NOT stInOuts.bTestFrameHomePos;
		I_PimSystem.mSetNewMachineState(nPIM_MachineStates._8_WaitForReset);
		iWorkStep := 91;
		
	91:	// Oczekiwanie na potwierdzenie
		IF I_PimSystem.mSetNewMachineState(nPIM_MachineStates._9_ResetInProgress) OR bServiceReset THEN
			fbTON_StepTimeout(IN:= FALSE);
			bServiceReset := FALSE;
			iWorkStep := 95;
		END_IF
		
	95:	// Potwierdzenie błedu
		IF NOT stInOuts.st2HandStartIO.bEmergButton_NC THEN
			mNewEvent(nEventClass:= nPIM_EventClasses.Error, nEvent:= nManometerCalibration_ErrorCodes.SafetySystemNotArmed);
		ELSE
			stInOuts.bNozzlePusherValve_Q := stInOuts.bTargetAirValve_Q := FALSE;
			IF stInOuts.bNozzlePusherHomePos THEN
				stInOuts.bTestFrameOpenValve_Q := FALSE;
				stInOuts.bTestFrameCloseValve_Q := TRUE;
				IF stInOuts.bTestFrameHomePos AND stInOuts.st2HandStartIO.bEmergButton_NC AND fbTON_StepTimeout.ET > T#200MS THEN
					nError := nManometerCalibration_ErrorCodes.NoError;
					I_PimSystem.mSetNewMachineState(nPIM_MachineStates._0_Standby_NotReady);
					iWorkStep := 0 ;	// Powrót do kroku inicjalizacyjnego lub wskazanego w algorytmie
				END_IF	
			END_IF
		END_IF
		fbTON_StepTimeout(IN:= TRUE, PT := T#4S);
		IF fbTON_StepTimeout.Q THEN
			mNewEvent(nEventClass:= nPIM_EventClasses.Error, nEvent:= nManometerCalibration_ErrorCodes.ResetTimeout);
		END_IF

	ELSE	// Krok domyślny w przypadku błędu w programie
		mNewEvent(nEventClass:= nPIM_EventClasses.Error, nEvent:= nManometerCalibration_ErrorCodes.ProgramConfigError);		
END_CASE

stInOuts.bNozzlePusherValve_Q R= stInOuts.bTargetAirValve_Q R= NOT stInOuts.st2HandStartIO.bEmergButton_NC;
stInOuts.bTestFrameCloseValve_Q R= stInOuts.bTestFrameOpenValve_Q R= NOT stInOuts.st2HandStartIO.bEmergButton_NC;

IF GVL_Aircom.stAC_DT_Data.bNew_Shift THEN
	udiNbOfSavedOkStatusesMEM:= udiNbOfSavedOkStatuses;
	udiNbOfSavedNokStatusesMEM := udiNbOfSavedNokStatuses;
	udiNbOfSavedOkStatuses := udiNbOfSavedNokStatuses := 0;
END_IF

METHOD FB_init : BOOL
VAR_INPUT
	bInitRetains : BOOL; // if TRUE, the retain variables are initialized (warm start / cold start)
	bInCopyCode : BOOL;  // if TRUE, the instance afterwards gets moved into the copy code (online change)
	I_Pim	: I_PIM;		// Interfejs do bloku PIM
END_VAR
I_PimSystem := I_Pim;
END_METHOD

(* Metoda TRUE kiedy dane wyjściowe są ok, jeśli nie FALSE (jeśli not bBusy i FALSE to błąd odczytu) *)
METHOD mGetParamsData : BOOL
VAR_INPUT
	bTestParams:	BOOL;	// Jeśli TRUE metoda okresla czy ma dostęp do parametrów, jeśli tak zwraca TRUE, jeśli nie FALSE
END_VAR
VAR_OUTPUT
	bBusy	: BOOL;										//	Maszyna odświeża dane
	pMachineParametersStruct	: POINTER TO BYTE;		// 	Wskaźnik do parametrów pracy maszyny
	uiMachineParametersSize	: UINT;						// 	Rozmiar struktury parametrów pracy maszyny [bajty]
	wActualCRC16SumInMachine	: WORD;					//	Aktualna suma CRC16 obliczona z parametrów
END_VAR
IF bTestParams THEN
	mGetParamsData := FALSE;
ELSE
	pMachineParametersStruct := 0;
	uiMachineParametersSize := 0;
	wActualCRC16SumInMachine := F_DATA_TO_CRC16_CCITT(pData := pMachineParametersStruct, cbData := uiMachineParametersSize, crc := 16#0000);
	bBusy := FALSE;
	mGetParamsData := TRUE;
END_IF
END_METHOD

METHOD INTERNAL mNewEvent : BOOL
VAR_INPUT
	nEventClass:nPIM_EventClasses;
	nEvent: nManometerCalibration_ErrorCodes;
END_VAR
IF nEventClass = nPIM_EventClasses.AlarmAutoConfirm OR nEventClass = nPIM_EventClasses.Message THEN		// Alarm nieblokadowy
	I_PimSystem.mSetNewMachineState(nPIM_MachineStates._0_Initialization);
	iWorkStep := 95;
ELSE
	I_PimSystem.mSetNewMachineState(nPIM_MachineStates._7_ErrorOccurr);
	I_PimSystem.mNewEvent(iEventId := nEvent, nEventType := nEventClass, tMessageTime := T#0S);
	iWorkStep := 90;
END_IF
nError := nEvent;
END_METHOD

END_FUNCTION_BLOCK

// ProdLineMachines/Sonictech/Fixtures/NoWeldLock/fbStFix_NoWeldLock
FUNCTION_BLOCK PUBLIC fbStFix_NoWeldLock EXTENDS fbStFixBaseTemplate IMPLEMENTS I_Fixture 
VAR_INPUT
	bEnclosureSensor:BOOL;
	bEnclosureSensoInvert:BOOL;
	bEnCheck:	BOOL;
END_VAR
VAR_OUTPUT
END_VAR
VAR
	fbEnclosureSensorFilter: fbBinaryFilter;
	bPartInFixture: BOOL;
	bPartWelded: BOOL;
	iCtr_SensorWorkVerification: INT;	// Value reset at every part pull up from fixture
END_VAR


fbEnclosureSensorFilter(IN := bEnclosureSensor XOR bEnclosureSensoInvert, tON := T#500MS, tOFF := T#500MS);
bPartInFixture S= fbEnclosureSensorFilter.RTrig;

IF fbEnclosureSensorFilter.FTrig THEN	// Wyjęcie części z kowadła
	IF bEnCheck AND bPartInFixture AND NOT bPartWelded THEN
		nQErrorId := nStFix_NoWeldLock_ErrorCodes.PartsNotWelded;
		iWorkStep := 90;
	END_IF
	bPartInFixture := bPartWelded := FALSE;
	iCtr_SensorWorkVerification := 0;	
END_IF

CASE iWorkStep OF
	0:		// Powrót do stanu początkowego (ustawienie zmiennych)
		bResetMethod := bQReady := bQBusy := bQError := FALSE;
		IF NOT bLock AND NOT bRelease THEN
			fbTON(IN:= FALSE);
			iWorkStep := 1;
		END_IF
			
	1: 		// Sprawdzenie czy siłowniki są w dobrej pozycji itp.
		bQLocked := FALSE;
		iWorkStep := 5;
	
	5:		// Oczekiwanie na nowy rozkaz
		bResetMethod:= bReleaseMethod:= bAuxOperMethod:= bLockMethod := FALSE;
		bQReady := TRUE;
		actCheckForNewOrder();
		
	10:		// Blokowanie kowadła
		IF iCtr_SensorWorkVerification > 2 THEN
			nQErrorId := nStFix_NoWeldLock_ErrorCodes.SensorWorkError;
			iWorkStep := 90;
		ELSE
			bQBusy := FALSE;
			nQErrorId := 0;
			iWorkStep := 5;				
		END_IF
		
	20:		// Dodatkowa operacja	
		bPartWelded:= bLastOperStatus;
		iCtr_SensorWorkVerification := iCtr_SensorWorkVerification +1;
		bQBusy := FALSE;
		iWorkStep := 5;

	30:	// Kowadło zwolnione
		bQBusy := FALSE;
		bQLocked := FALSE;		
		iWorkStep := 5;
		
	50:	// Manual mode
		bManualWork :=FALSE;
		iWorkStep := 5;
		
	90:		// Błąd w pracy kowadła
		bQBusy := FALSE;
		bQError := TRUE;
		iWorkStep := 91;
		
	91:
		IF bRelease OR bResetMethod THEN
			iCtr_SensorWorkVerification := 0;
			bPartInFixture := bPartWelded := FALSE;
			bQError := FALSE;
			nQErrorId := iWorkStep := 0;
		END_IF
		
END_CASE

END_FUNCTION_BLOCK

// ProdLineMachines/Sonictech/Fixtures/fbStFixBaseTemplate
// Dont change this!!!
FUNCTION_BLOCK PUBLIC fbStFixBaseTemplate IMPLEMENTS I_Fixture
VAR_INPUT
	bLock			: BOOL;
	bAuxOper		: BOOL;
	bRelease		: BOOL;
END_VAR
VAR_OUTPUT
	bQReady			: BOOL;		// GOtowość na kolejny rozkaz
	bQBusy			: BOOL;		// Kowadło w ruchu (blokowanie lub odblokowanie trwa)
	bQLocked		: BOOL;		// Kowadło zablokowane (jeśli false i Ready TRUE to odblokowane)
	bQError			: BOOL;		// Błąd w pracy
	nQErrorId		: INT;		// Error Code
END_VAR
VAR
	iWorkStep: INT;
	nMachActState: nPIM_MachineStates;
	bManualWork, bLastOperStatus, bTestMode, bUserLogged, bWeldingActive: BOOL;
	fbTON: TON;				// Timeout timer
	bResetMethod, bReleaseMethod, bAuxOperMethod, bLockMethod: BOOL;	// Orders from method calls
	bTestOutputs: BOOL;			// When True outputs is tested in manual mode
	fbFTRIG_TestOutputs: F_TRIG;	// Testing of outputs ended - reset to base state
END_VAR

fbFTRIG_TestOutputs(CLK:= bTestOutputs); 

CASE iWorkStep OF
	0:		// Return to the base state (Variables set)
		bResetMethod := bQReady := bQBusy := bQError := FALSE;
		IF NOT bLock AND NOT bRelease THEN
			fbTON(IN:= FALSE);
			iWorkStep := 1;
		END_IF
			
	1: 		// Check if pistons are in desired positions etc.
		fbTON(IN:= TRUE, PT:= T#2S);
		bQLocked := FALSE;
		iWorkStep := 5;
	
	5:		// Waiting for new order
		bQReady := TRUE;
		actCheckForNewOrder();
		
	10:		// Locking of the part in the fixture
		bQLocked := TRUE;		
		iWorkStep := 5;
	
	30:		// Release part
		bQLocked := FALSE;		
		iWorkStep := 5;
		
	50:		// Manual work coordination
		fbTON(IN:= TRUE, PT:= T#15M);
		IF NOT bManualWork OR fbTON.Q THEN
			fbTON(IN:= FALSE);
			bManualWork := FALSE;
			iWorkStep := 0;
		END_IF
		
	90:		// Fixture work error
		bQBusy := FALSE;
		bQReady := bQError := TRUE;
		IF bRelease OR bResetMethod THEN
			bQError := FALSE;
			nQErrorId := iWorkStep := 0;
		END_IF
END_CASE

// Fixture in error state - reset required
PROPERTY prFixError : BOOL
GET
prFixError := bQError;
END_GET
END_PROPERTY

// Active/last error code
PROPERTY prFixErrorID : INT
GET
prFixErrorID := nQErrorId;
END_GET
END_PROPERTY

// Is fixture is locked (part is locked)
PROPERTY prFixLocked : BOOL
GET
prFixLocked := bQLocked AND NOT bQBusy AND bQReady;
END_GET
END_PROPERTY

// Fixture redy for new operation
PROPERTY prFixReady : BOOL
GET
prFixReady := bQReady;
END_GET
END_PROPERTY

// Fixture released (part is unlocked)
PROPERTY prFixReleased : BOOL
GET
prFixReleased := NOT bQLocked AND NOT bQBusy AND bQReady;
END_GET
END_PROPERTY

// Machine state of us welder
PROPERTY prMachState : nPIM_MachineStates
SET
nMachActState := prMachState;
END_SET
END_PROPERTY

// Is test mode active
PROPERTY prTestMode : BOOL
SET
bTestMode := prTestMode;
END_SET
END_PROPERTY

// Ultrasonic generation active (welding active)
PROPERTY prTestOutputsActive : BOOL
SET
bTestOutputs:= prTestOutputsActive;
END_SET
END_PROPERTY

// Is user logged in
PROPERTY prUserLogged : BOOL
SET
bUserLogged:= prUserLogged;
END_SET
END_PROPERTY

// Ultrasonic generation active (welding active)
PROPERTY prWeldingActive : BOOL
SET
bWeldingActive := prWeldingActive;
END_SET
END_PROPERTY

ACTION actCheckForNewOrder:
// Checking if there is new order
IF bLock OR bLockMethod THEN
	iWorkStep := 10;
ELSIF bAuxOper OR bAuxOperMethod THEN
	iWorkStep := 20;
ELSIF bRelease OR bReleaseMethod THEN
	iWorkStep := 30;		
ELSIF bManualWork THEN
	iWorkStep := 50;			
END_IF
IF iWorkStep <> 5 THEN
	fbTON(IN:= FALSE);
	bQReady := FALSE;
	bQBusy := TRUE;
END_IF
END_ACTION

// Wysłanie rozkazu do wykonania na części w kowadle dodatkowej operacji po zakończeniu operacji, zwraca true gdy można odczytać wynik operacji
METHOD mAuxOper : BOOL
VAR_INPUT
	bOperStatus: BOOL;	// Status operacji
END_VAR
VAR_OUTPUT
	bBusy:	BOOL;		// Flaga pracy kowadła
	bError:	BOOL;		// Flaga błędu podczas blokowania
	nErrorCode: INT;	// Kod błędu
END_VAR
IF bQReady THEN
	bLastOperStatus:= bOperStatus;
	bAuxOperMethod := TRUE;
	actCheckForNewOrder();
	bBusy := bQBusy;
ELSIF bAuxOperMethod THEN
	IF bQBusy THEN
		bBusy := TRUE;
	ELSE
		mAuxOper := TRUE;
		bAuxOperMethod := bBusy := FALSE;
		bError := bQError;
		nErrorCode:= nQErrorId;
	END_IF
ELSE
	mAuxOper := bBusy := FALSE;
END_IF
END_METHOD

// Wysłanie rozkazu do zablokowania części w kowadle, zwraca true gdy można odczytać wynik operacji
METHOD mLock : BOOL
VAR_OUTPUT
	bBusy:	BOOL;		// Flaga pracy kowadła
	bError:	BOOL;		// Flaga błędu podczas blokowania
	nErrorCode: INT;	// Kod błędu
END_VAR
IF bQReady THEN
	bLockMethod := TRUE;
	actCheckForNewOrder();
	bBusy := bQBusy;
ELSIF bLockMethod THEN
	IF bQBusy THEN
		bBusy := TRUE;
	ELSE
		mLock := TRUE;
		bLockMethod := bBusy := FALSE;
		bError := bQError;
		nErrorCode:= nQErrorId;
	END_IF
ELSE
	mLock := bBusy := FALSE;
END_IF
END_METHOD

METHOD PROTECTED mNewEvent
VAR_INPUT
	nErrID: INT;
END_VAR
bLock := bRelease := bAuxOper := FALSE;
bQError := TRUE;
nQErrorId := nErrID;
iWorkStep := 90;
END_METHOD

// Rozkaz do odblokowania części w kowadle, zwraca true gdy można odczytać wynik operacji
METHOD mRelease : BOOL
VAR_INPUT
	bReset:BOOL;		// Reset kowadła do stanu spoczynku (z dowolnego stanu)
END_VAR
VAR_OUTPUT
	bBusy:	BOOL;		// Flaga pracy kowadła
	bError:	BOOL;		// Flaga błędu podczas odblokowania
	nErrorCode: INT;	// Kod błędu
END_VAR
IF bReset THEN
	iWorkStep := 0;
	bBusy := bError := FALSE;
	mRelease := TRUE;
ELSIF bQError THEN
	bResetMethod := TRUE;
ELSIF bQReady THEN
	bReleaseMethod := TRUE;
	actCheckForNewOrder();
	bBusy := bQBusy;
ELSIF bReleaseMethod THEN
	IF bQBusy THEN
		bBusy := TRUE;
	ELSE
		mRelease := TRUE;
		bReleaseMethod := bBusy := FALSE;
		bError := bQError;
		nErrorCode:= nQErrorId;
	END_IF
ELSE
	mRelease := bBusy := FALSE;
END_IF
END_METHOD

END_FUNCTION_BLOCK

// ProdLineMachines/Sonictech/Fixtures/I_Fixture
INTERFACE I_Fixture

// Fixture in error state - reset required
PROPERTY prFixError : BOOL
GET
END_GET
END_PROPERTY

// Active/last error code
PROPERTY prFixErrorID : INT
GET
END_GET
END_PROPERTY

// Is fixture is locked (part is locked)
PROPERTY prFixLocked : BOOL
GET
END_GET
END_PROPERTY

// Fixture redy for new operation
PROPERTY prFixReady : BOOL
GET
END_GET
END_PROPERTY

// Fixture released (part is unlocked)
PROPERTY prFixReleased : BOOL
GET
END_GET
END_PROPERTY

// Machine state of us welder
PROPERTY prMachState : nPIM_MachineStates
SET
END_SET
END_PROPERTY

// Is test mode active
PROPERTY prTestMode : BOOL
SET
END_SET
END_PROPERTY

// Ultrasonic generation active (welding active)
PROPERTY prTestOutputsActive : BOOL
SET
END_SET
END_PROPERTY

// Is user logged in
PROPERTY prUserLogged : BOOL
SET
END_SET
END_PROPERTY

// Ultrasonic generation active (welding active)
PROPERTY prWeldingActive : BOOL
SET
END_SET
END_PROPERTY

// Wysłanie rozkazu do wykonania na części w kowadle dodatkowej operacji po zakończeniu operacji, zwraca true gdy można odczytać wynik operacji
METHOD mAuxOper : BOOL
VAR_INPUT
	bOperStatus: BOOL;	// Status operacji
END_VAR
VAR_OUTPUT
	bBusy:	BOOL;		// Flaga pracy kowadła
	bError:	BOOL;		// Flaga błędu podczas blokowania
	nErrorCode: INT;	// Kod błędu
END_VAR
END_METHOD

// Wysłanie rozkazu do zablokowania części w kowadle, zwraca true gdy można odczytać wynik operacji
METHOD mLock : BOOL
VAR_OUTPUT
	bBusy:	BOOL;		// Flaga pracy kowadła
	bError:	BOOL;		// Flaga błędu podczas blokowania
	nErrorCode: INT;	// Kod błędu
END_VAR
END_METHOD

// Rozkaz do odblokowania części w kowadle, zwraca true gdy można odczytać wynik operacji
METHOD mRelease : BOOL
VAR_INPUT
	bReset:BOOL;		// Reset kowadła do stanu spoczynku (z dowolnego stanu)
END_VAR
VAR_OUTPUT
	bBusy:	BOOL;		// Flaga pracy kowadła
	bError:	BOOL;		// Flaga błędu podczas odblokowania
	nErrorCode: INT;	// Kod błędu
END_VAR
END_METHOD

END_INTERFACE

// ProdLineMachines/Sonictech/Fixtures/S01_IndicatorAssembly/fbStFix_S01IndicatorAssy
FUNCTION_BLOCK PUBLIC fbStFix_S01IndicatorAssy EXTENDS fbStFixBaseTemplate IMPLEMENTS I_Fixture 
VAR_IN_OUT
	stInOuts:stStFix_S01IndicatorAssy_InOut;
END_VAR
VAR_INPUT
	stTestParams:stStFix_S01IndicatorAssy_Settings;
	iMaxTrigRepeats: INT := 3;
END_VAR
VAR_OUTPUT
END_VAR
VAR
	fbBVS: fbBvsControl;
	I_Vision: I_VisionSensorSTD;
	iTriggerRepeats: INT;
	bErrorBVS: BOOL;
	bIndicator, bVring, bCap: BOOL;		// WYnik detekcji	
END_VAR

fbBVS(stIO_Data:= stInOuts.stBalluff, tMinImpWidth:= T#30MS);
I_Vision := fbBVS;

stInOuts.bVacuumON_Q := bUserLogged AND stTestParams.bVacumEN;

CASE iWorkStep OF
	0:		// Powrót do stanu początkowego (ustawienie zmiennych)
		bResetMethod := bQReady := bQBusy := bQError := FALSE;
		fbBVS.bTrigger := FALSE;
		IF NOT bLock AND NOT bRelease THEN
			fbTON(IN:= FALSE);
			iWorkStep := 1;
		END_IF
			
	1: 		// Sprawdzenie czy siłowniki są w dobrej pozycji itp.
		fbTON(IN:= TRUE, PT:= T#2S);
		bQLocked := FALSE;
		iWorkStep := 5;
	
	5:		// Oczekiwanie na nowy rozkaz
		bResetMethod:= bReleaseMethod:= bAuxOperMethod:= bLockMethod := FALSE;
		bQReady := TRUE;
		actCheckForNewOrder();	
		
	10:		// Blokowanie kowadła
		nQErrorId := iTriggerRepeats := 0;
		iWorkStep := 12;
		
	12:		// Oczekiwanie na zakończenie detekcji
		IF I_Vision.mNewInspection(bError => bErrorBVS, bOut1=> bIndicator, bOut2=>bVring, bOut3 => bCap) THEN
			IF NOT bErrorBVS THEN		// Balluff odpowiedział
				IF (bIndicator OR NOT stTestParams.bIndicatorCheckEN) AND (bVring OR NOT stTestParams.bVRingCheckEN) AND (bCap OR NOT stTestParams.bCapCheckEN) THEN		// Wszystko wykryte
					iWorkStep := 16;
				ELSE		// NIe wyszystko wykryte
					IF iTriggerRepeats >= iMaxTrigRepeats THEN		// Wykonano powtórne zdjęcie
						IF NOT bIndicator AND bVring AND bCap THEN
							mNewEvent(nStFix_S01IndicatorAssy_ErrorCodes.IndicatorNotDet);

						ELSIF bIndicator AND NOT bVring AND bCap THEN
							mNewEvent(nStFix_S01IndicatorAssy_ErrorCodes.VRingNotDet);
						ELSIF NOT bIndicator AND NOT bVring AND bCap THEN
							mNewEvent(nStFix_S01IndicatorAssy_ErrorCodes.VRingIndicatorNotDet);
						ELSIF bIndicator AND bVring AND NOT bCap THEN
							mNewEvent(nStFix_S01IndicatorAssy_ErrorCodes.CapNotDet);
						ELSIF NOT bIndicator AND bVring AND NOT bCap THEN
							mNewEvent(nStFix_S01IndicatorAssy_ErrorCodes.CapIndicatorNotDet);	
						ELSIF bIndicator AND NOT bVring AND NOT bCap THEN
							mNewEvent(nStFix_S01IndicatorAssy_ErrorCodes.CapVRingNotDet);	
						ELSIF NOT bIndicator AND NOT bVring AND NOT bCap THEN
							mNewEvent(nStFix_S01IndicatorAssy_ErrorCodes.CapVRingIndicatorNotDet);	
						END_IF
					ELSE		// Wykonaj powtórne zdjęcie
						iTriggerRepeats := iTriggerRepeats + 1;
						fbTON(IN:= FALSE);
						iWorkStep := 14;
					END_IF
				END_IF
			ELSE		// brak odpowiedzi Balluffa
				mNewEvent(nStFix_S01IndicatorAssy_ErrorCodes.SensorNotReady);
			END_IF
		END_IF
		
	14:		// Oczekiwanie oraz powtórna próba znalezienia
		fbTON(IN:= TRUE, PT:= T#200MS);
		IF fbTON.Q THEN
			fbTON(IN:= FALSE);
			iWorkStep := 12;
		END_IF
	16:		// Wszystko wykryte OK
		bLock := bQError := bQBusy := FALSE;
		iWorkStep := 5;
	
	20:		// Dodatkowa operacja
		bAuxOper := bQBusy := FALSE;
		bQLocked := FALSE;		
		iWorkStep := 5;
	
	30:		// Zwalnianie kowadła
		bRelease := bQBusy := bQLocked := FALSE;		
		iWorkStep := 5;

	50:		// Manual work coordination
		fbTON(IN:= TRUE, PT:= T#15M);
		IF NOT bManualWork OR fbTON.Q THEN
			fbTON(IN:= FALSE);
			bManualWork := FALSE;
			iWorkStep := 0;
		END_IF
		
	90:		// Błąd w pracy kowadła
		bQBusy := FALSE;
		bQError := TRUE;
		fbBVS.bTrigger := fbBVS.bReadActualInspection := fbBVS.bChangeInspection := FALSE;
		iWorkStep := 91;
		
	91:
		IF bRelease OR bResetMethod THEN
			bQError := FALSE;
			nQErrorId := iWorkStep := 0;
		END_IF

	ELSE
		mNewEvent(nStFix_S01IndicatorAssy_ErrorCodes.ProgramConfigError);		
END_CASE

END_FUNCTION_BLOCK

// VisionSensors/Balluff BVS/fbBvsControl
FUNCTION_BLOCK fbBvsControl IMPLEMENTS I_VisionSensorSTD
VAR_IN_OUT
	stIO_Data: stBVS_DigInOut;
END_VAR
VAR_INPUT
	bTrigger:BOOL;
	bReadActualInspection:BOOL;
	bChangeInspection:BOOL;		// Zbocze narastające inicjuje zmianę programu
	iInspectionToActive:INT;
	tMinImpWidth:TIME;		// Czas minimalnego trwania impulsu
END_VAR
VAR_OUTPUT
	bBusy: BOOL;
	bOutput1: BOOL;
	bOutput2: BOOL;
	bOutput3: BOOL;
	bError:	BOOL;
	bResultReady: BOOL;
	iActiveProgramId:INT;
END_VAR
VAR
	iWorkStep:INT;
	fbTP_ImpuleGen:TP;
	wConfirmedDeterctionNumber: WORD;
	fbTON_Timeout: TON;
	bToggleMemory: BOOL;
	bNewInspectionBusy :BOOL;
	fbTON_CmdTimeout: TON;
	bReadInspectionBusy: BOOL;
	bSetInspectionBusy: BOOL;
	iIdToSet: INT;
	fbTON_NewStep: TON;
	fbTP_ImpulesRead: TP;
	fbTON_NewStepLong: TON;
	iTargetIdToSet: INT;
END_VAR

IF iWorkStep > 10 THEN
	fbTP_ImpuleGen(IN:= FALSE, PT:= tMinImpWidth + T#5MS);	
	fbTP_ImpulesRead(IN:= FALSE, PT:= 2*tMinImpWidth);	
	fbTON_NewStep(IN:= TRUE,PT:= tMinImpWidth);
	fbTON_NewStepLong(IN:= TRUE,PT:= 2*tMinImpWidth);
	IF iWorkStep < 90 THEN
		fbTON_CmdTimeout(IN:= TRUE, PT:= T#7S);
		IF fbTON_CmdTimeout.Q THEN
			fbTON_CmdTimeout(IN:= FALSE);
			iWorkStep := 90;
		END_IF
	END_IF	
END_IF


CASE iWorkStep OF
	0:	// Inicjalizacja
		stIO_Data.bDO_InputSelect:= stIO_Data.bDO_Trigger:= FALSE;
		fbTON_Timeout(IN:= FALSE);
		iWorkStep := 5;
	
	5:	// Oczekiwanie na rozkazy
		IF bNewInspectionBusy OR bTrigger THEN		// Nowa detekcja
			bBusy := TRUE;
			bError := bSetInspectionBusy := bReadInspectionBusy := bOutput1 := bOutput2 := bOutput3 := bResultReady := FALSE;
			stIO_Data.bDO_Trigger := TRUE;
			bToggleMemory:= stIO_Data.bDI_TriggerSignal;
			fbTON_CmdTimeout(IN:= FALSE);
			iWorkStep := 10;
		ELSIF bReadInspectionBusy OR bReadActualInspection THEN		// Odczyt Id detekcji
			bBusy := TRUE;
			bError := bSetInspectionBusy := bResultReady := FALSE;
			iIdToSet := 21;
			iActiveProgramId := -1;
			fbTON_CmdTimeout(IN:= FALSE);
			iWorkStep := 20;
		ELSIF bSetInspectionBusy OR bChangeInspection THEN			// Ustawienie nowej detekcji
			IF bChangeInspection THEN
				IF iInspectionToActive > 0 AND iInspectionToActive <= 20 THEN
					iIdToSet := iInspectionToActive;
				END_IF		
			END_IF
			IF iIdToSet > 0 AND iIdToSet <= 20 THEN 			
				bBusy := TRUE;
				bError := bResultReady := FALSE;
				iTargetIdToSet:= iIdToSet;
				iActiveProgramId := -1;
				fbTON_CmdTimeout(IN:= FALSE);
				iWorkStep := 20;
			ELSE	
				bBusy := FALSE;
				bError := bResultReady := TRUE;
				iActiveProgramId := -1;
				iWorkStep := 6;
			END_IF
		END_IF
		
	6:	// Oczekiwanie po wykonanej komendzie na sygnał zerowy na poszczególnych wejściach
		IF NOT bTrigger AND NOT bReadActualInspection AND NOT bChangeInspection THEN
			fbTON_Timeout(IN:= TRUE, PT:= T#1S);
			IF (NOT bNewInspectionBusy AND NOT bReadInspectionBusy AND NOT bSetInspectionBusy) OR fbTON_Timeout.Q THEN
				bNewInspectionBusy := bReadInspectionBusy := bSetInspectionBusy := FALSE;
				bBusy := stIO_Data.bDO_Trigger := stIO_Data.bDO_InputSelect := FALSE;
				fbTON_CmdTimeout(IN:= FALSE);
				fbTON_Timeout(IN:= FALSE);
				iWorkStep := 0;
			END_IF	
		END_IF
	
	10:	// Detekcja wyzwolona, oczekiwanie na rezultat
		fbTON_CmdTimeout(IN:= TRUE, PT:= T#500MS);
		IF bToggleMemory <> stIO_Data.bDI_TriggerSignal THEN		// Detekcja zakończona
			bOutput1 := stIO_Data.bDI_Input_1;
			bOutput2 := stIO_Data.bDI_Input_2;
			bOutput3 := stIO_Data.bDI_Input_3;
			bResultReady := TRUE;
			bBusy := FALSE;
			bToggleMemory := stIO_Data.bDI_TriggerSignal;
			stIO_Data.bDO_Trigger := FALSE;
			iWorkStep := 6;
		ELSIF fbTON_CmdTimeout.Q THEN
			bBusy := FALSE;
			bError := TRUE;
			stIO_Data.bDO_Trigger := FALSE;
			iWorkStep := 6;
		END_IF
		IF iWorkStep <> 10 THEN fbTON_Timeout(IN:= FALSE); fbTON_CmdTimeout(IN:= FALSE); END_IF
				
		
	20:	// Odczyt/zmiana aktywnego programu 
		stIO_Data.bDO_Trigger := stIO_Data.bDO_InputSelect := FALSE;
		fbTON_NewStep(IN:= FALSE);
		iWorkStep := 21;
	21:	// ***** FAZA 1 ***** Ustawienie sygnału wyboru programu	
		IF fbTON_NewStep.Q THEN
			stIO_Data.bDO_InputSelect := TRUE;
			fbTON_NewStep(IN:= FALSE);
			iWorkStep := 22;
		END_IF	
	22:	// ***** FAZA 2 ***** Oczekiwanie na wygaszenie wyjść i generacja impulsu
		IF NOT stIO_Data.bDI_Input_1 AND NOT stIO_Data.bDI_Input_2 AND NOT stIO_Data.bDI_Input_3 AND fbTON_NewStep.Q THEN
			fbTP_ImpuleGen(IN:= NOT stIO_Data.bDO_Trigger);
			stIO_Data.bDO_Trigger := fbTP_ImpuleGen.Q;
			iWorkStep := 23;	
		END_IF
	23:
		stIO_Data.bDO_Trigger := fbTP_ImpuleGen.Q;
		IF NOT stIO_Data.bDO_Trigger THEN
			fbTON_NewStep(IN:= FALSE);
			iWorkStep := 24;	
		END_IF	
	24:	// ***** FAZA 3 ***** Oczekiwanie na wystawienie wyjść
		IF stIO_Data.bDI_Input_1 AND stIO_Data.bDI_Input_2 AND stIO_Data.bDI_Input_3 AND fbTON_NewStep.Q THEN
			fbTON_NewStep(IN:= FALSE);
			iWorkStep := 25;	
		END_IF
	25:	// ***** FAZA 3 ***** Generacja liczby impulsów odpowiadających numerowi detekcji
		IF iIdToSet > 0 THEN
			iWorkStep := 26;
		ELSE
			fbTON_NewStep(IN:= FALSE);
			iWorkStep := 27;
		END_IF
	26:	// ***** FAZA 3 ***** Generacja liczby impulsów odpowiadających numerowi detekcji
		fbTP_ImpuleGen(IN:= NOT stIO_Data.bDO_Trigger);
		stIO_Data.bDO_Trigger := fbTP_ImpuleGen.Q;
		IF NOT stIO_Data.bDO_Trigger THEN
			iIdToSet := iIdToSet -1;
			fbTON_NewStep(IN:= FALSE);
			iWorkStep := 27;
		END_IF
	27:	// ***** FAZA 3 ***** Pauza pomiędzy impulsami
		IF fbTON_NewStep.Q THEN
			IF iIdToSet > 0 THEN
				iWorkStep := 25;
			ELSE
				iWorkStep := 28;
			END_IF
		END_IF
	28:	// ***** FAZA 4 ***** Kasowanie sygnału ustawienia inspekcji
		stIO_Data.bDO_Trigger := stIO_Data.bDO_InputSelect := FALSE;
		IF NOT stIO_Data.bDI_Input_1 AND NOT stIO_Data.bDI_Input_2 AND NOT stIO_Data.bDI_Input_3 THEN
			fbTON_NewStep(IN:= FALSE);
			iWorkStep := 29;
		END_IF
	29:	// Wystawienie pierwszego sygnału trigger
		IF fbTON_NewStep.Q THEN
			fbTP_ImpulesRead(IN:= NOT stIO_Data.bDO_Trigger);
			stIO_Data.bDO_Trigger := fbTP_ImpulesRead.Q;
			IF NOT stIO_Data.bDO_Trigger THEN
				wConfirmedDeterctionNumber.0 := stIO_Data.bDI_Input_1;
				wConfirmedDeterctionNumber.1 := stIO_Data.bDI_Input_2;
				wConfirmedDeterctionNumber.2 := stIO_Data.bDI_Input_3;
				fbTON_NewStepLong(IN:= FALSE);
				iWorkStep := 30;
			END_IF
		END_IF
		
	30:
		IF NOT stIO_Data.bDI_Input_1 AND NOT stIO_Data.bDI_Input_2 AND NOT stIO_Data.bDI_Input_3 AND fbTON_NewStepLong.Q THEN
			fbTON_NewStep(IN:= FALSE);
			iWorkStep := 31;
		END_IF
	31:
		IF fbTON_NewStep.Q THEN
			fbTP_ImpulesRead(IN:= NOT stIO_Data.bDO_Trigger);
			stIO_Data.bDO_Trigger := fbTP_ImpulesRead.Q;
			IF NOT stIO_Data.bDO_Trigger THEN
				wConfirmedDeterctionNumber.3 := stIO_Data.bDI_Input_1;
				wConfirmedDeterctionNumber.4 := stIO_Data.bDI_Input_2;
				wConfirmedDeterctionNumber.5 := stIO_Data.bDI_Input_3;
				fbTON_NewStepLong(IN:= FALSE);
				iWorkStep := 32;
			END_IF
		END_IF
	32:
		IF NOT stIO_Data.bDI_Input_1 AND NOT stIO_Data.bDI_Input_2 AND NOT stIO_Data.bDI_Input_3 AND fbTON_NewStepLong.Q THEN
			fbTON_NewStep(IN:= FALSE);
			iWorkStep := 33;
		END_IF
	33:
		IF fbTON_NewStep.Q THEN
			fbTP_ImpuleGen(IN:= NOT stIO_Data.bDO_Trigger);
			stIO_Data.bDO_Trigger := fbTP_ImpuleGen.Q;
			IF NOT stIO_Data.bDO_Trigger THEN
				iWorkStep := 34;
			END_IF
		END_IF
	34:
		IF NOT stIO_Data.bDI_Input_1 AND NOT stIO_Data.bDI_Input_2 AND NOT stIO_Data.bDI_Input_3 THEN
			bBusy := FALSE;
			iActiveProgramId := WORD_TO_INT(wConfirmedDeterctionNumber);
			bResultReady := TRUE;
			bError := iTargetIdToSet = iActiveProgramId;
			iWorkStep := 1;
		END_IF
			
	90:	// In case of error ...
		bError := TRUE;
		bBusy := FALSE;
		stIO_Data.bDO_Trigger := stIO_Data.bDO_InputSelect := FALSE;
		fbTON_CmdTimeout(IN:= TRUE, PT:= T#2S);
		IF fbTON_CmdTimeout.Q THEN
			iWorkStep := 1; 
		END_IF

END_CASE

METHOD mNewInspection : BOOL (* Metoda zwraca true gdy detekcja zostanie zakończona*)
VAR_OUTPUT
	bError	: BOOL;			// Informacja zakończeniu detekcji z błędem
	bOut1, bOut2, bOut3, bOut4	: BOOL;		// Wyjścia zostają odświeżone po zakońcoznej detekcji 
END_VAR
IF iWorkStep = 5 THEN
	bOut1 := bOut2 := bOut3 := bOut4 := bResultReady := FALSE;
	bNewInspectionBusy := TRUE;
ELSIF bNewInspectionBusy THEN
	IF bResultReady THEN
		bOut1 := bOutput1;
		bOut2 := bOutput2;
		bOut3 := bOutput3;
		bNewInspectionBusy := bError := bOut4 := FALSE;
		mNewInspection := TRUE;
	ELSIF fbTON_CmdTimeout.Q THEN
		bError := mNewInspection := TRUE;	
		bNewInspectionBusy := FALSE;
	END_IF
ELSE
	bError := mNewInspection := TRUE;
END_IF
END_METHOD

METHOD mReadInspectionId : BOOL (* Metoda zwraca true gdy zakończyła pracę*)
VAR_OUTPUT
	bError	: BOOL;			// Błąd ustawienia
	iActiveInspectionId	: INT;		// Identyfikator aktualnej inspekcji
END_VAR
IF iWorkStep = 0 THEN
	bResultReady := FALSE;
	bReadInspectionBusy := TRUE;
ELSIF bReadInspectionBusy THEN
	IF bResultReady THEN
		bReadInspectionBusy := bError := FALSE;
		iActiveInspectionId := iActiveProgramId;
		mReadInspectionId := TRUE;
	ELSIF fbTON_CmdTimeout.Q THEN
		bError := mReadInspectionId := TRUE;	
		iActiveInspectionId := -1;
		bReadInspectionBusy := FALSE;
	END_IF
ELSE
	bError := mReadInspectionId := TRUE;
	iActiveInspectionId := -1;
END_IF
END_METHOD

METHOD mSetInspectionId : BOOL
VAR_OUTPUT
	bError	: BOOL; 		// Błąd ustawienia
	iActiveInspectionId	: INT;		// Identyfikator aktualnej inspekcji
END_VAR
VAR_INPUT
	iInspectionIdToSet	: INT;			// Identyfikator inspekcji do ustawienia
END_VAR
IF iWorkStep = 0 AND iInspectionIdToSet <= 20 AND iInspectionIdToSet > 0 THEN
	bResultReady := FALSE;
	iIdToSet := iInspectionIdToSet;
	bSetInspectionBusy := TRUE;
ELSIF bSetInspectionBusy THEN
	IF bResultReady THEN
		bSetInspectionBusy := bError := FALSE;
		bError := iActiveProgramId <> iInspectionIdToSet;
		iActiveInspectionId := iActiveProgramId;
		mSetInspectionId := TRUE;
	ELSIF fbTON_CmdTimeout.Q THEN
		bError := mSetInspectionId := TRUE;	
		iActiveInspectionId := -1;
		bSetInspectionBusy := FALSE;
	END_IF
ELSE
	bError := mSetInspectionId := TRUE;
	iActiveInspectionId := -1;
END_IF
END_METHOD

END_FUNCTION_BLOCK

// VisionSensors/I_VisionSensorSTD
INTERFACE I_VisionSensorSTD

METHOD mNewInspection : BOOL	// Metoda zwraca true gdy detekcja zostanie zakończona
VAR_OUTPUT
	bError: BOOL;		// Informacja zakończeniu detekcji z błędem
	bOut1, bOut2, bOut3, bOut4: BOOL;	// Po zakońcoznej detekcji wyjścia zostają odświeżone
END_VAR

VAR_INPUT
END_VAR
END_METHOD

METHOD mReadInspectionId : BOOL			// Metoda zwraca true gdy zakończyła pracę
VAR_OUTPUT
	bError: BOOL;						// Błąd ustawienia
	iActiveInspectionId:INT;			// Identyfikator aktualnej inspekcji
END_VAR
VAR_INPUT
END_VAR
END_METHOD

METHOD mSetInspectionId : BOOL
VAR_OUTPUT
	bError: BOOL;						// Błąd ustawienia
	iActiveInspectionId	: INT;		// Identyfikator aktualnej inspekcji
END_VAR
VAR_INPUT
	iInspectionIdToSet:INT;				// Identyfikator inspekcji do ustawienia
END_VAR
END_METHOD

END_INTERFACE

// ProdLineMachines/Sonictech/Fixtures/S06_CarrierWheelLubrification/V1/fbStFix_S06CarrierAndWheelAssyGrease
FUNCTION_BLOCK PUBLIC fbStFix_S06CarrierAndWheelAssyGrease EXTENDS fbStFixBaseTemplate IMPLEMENTS I_Fixture 
VAR_IN_OUT
	stInOuts:stStFix_S06CarrierAndWheelAssyGrease_InOuts;
END_VAR
VAR_INPUT
	// Wejścia cyfrowe, konfiguracyjne itp
	stSettings : stStFix_S06CarrierAndWheelAssyGrease_Settings;
END_VAR
VAR_OUTPUT
	// Wyjścia cyfrowe itp
END_VAR
VAR
	fbTP_Grease: TP;
	fbTOF_Delay: TOF;
END_VAR

fbTP_Grease(IN:= FALSE, PT:= REAL_TO_TIME(stSettings.rGreaseApplyTime*1000), Q=> stInOuts.bGreaseValve_Q);

CASE iWorkStep OF
	0:		// Powrót do stanu początkowego (ustawienie zmiennych)
		bResetMethod := bQReady := bQBusy := bQError := FALSE;
		IF NOT bLock AND NOT bRelease THEN
			fbTON(IN:= FALSE);
			iWorkStep := 1;
		END_IF
			
	1: 		// Sprawdzenie czy siłowniki są w dobrej pozycji itp.
		stInOuts.bRotationStabValve_Q := stInOuts.bNozzleStabValve_Q := stInOuts.bGreaseValve_Q := FALSE;
		bQLocked := FALSE;
		fbTON(IN:= FALSE);
		iWorkStep := 5;
	
	5:		// Oczekiwanie na nowy rozkaz
		bQReady := TRUE;
		bResetMethod:= bReleaseMethod:= bAuxOperMethod:= bLockMethod := FALSE;
		actCheckForNewOrder();
		
	10:		// Blokowanie kowadła
		fbTON(IN:= TRUE, PT:= T#700MS);
		stInOuts.bRotationStabValve_Q := TRUE;
		IF stInOuts.bRotationStabilizerClosed THEN
			iWorkStep := 12;
		ELSIF fbTON.Q THEN
			nQErrorId := nStFix_S06CarrierAndWheelAssyGrease_ErrorCodes.StabilizingTimeout;
			iWorkStep := 90;
		END_IF
		IF iWorkStep <> 10 THEN fbTON(IN:= FALSE); END_IF
  
	12:		// Oczekiwanie na zakończenie detekcji
		fbTON(IN:= TRUE, PT:= T#500MS);
		stInOuts.bNozzleStabValve_Q := TRUE;
		IF NOT stInOuts.bNozzleStabilizerClosed THEN
			iWorkStep := 14;
		ELSIF fbTON.Q THEN
			nQErrorId := nStFix_S06CarrierAndWheelAssyGrease_ErrorCodes.StabilizingTimeout;	
			iWorkStep := 90;
		END_IF
		IF iWorkStep <> 12 THEN fbTON(IN:= FALSE); END_IF
		
	14:		// Wszystko  OK
		bQBusy := FALSE;		
		bQLocked := TRUE;		
		iWorkStep := 5;
		
	20: 	// Dodatkowa operacja - smarowanie
		IF bLastOperStatus THEN
			fbTP_Grease(IN:= TRUE);	
			bQBusy := FALSE;		
			iWorkStep := 5;
		ELSE
			bQError := bQBusy := FALSE;	
		END_IF
		fbTOF_Delay(IN:= FALSE);
		
	30:		// Zwalnianie kowadła
		fbTON(IN:= TRUE, PT:= T#1500MS);
		fbTOF_Delay(IN:= stInOuts.bGreaseValve_Q, PT:= T#150MS);
		stInOuts.bNozzleStabValve_Q := fbTOF_Delay.Q;
		IF stInOuts.bNozzleStabilizerClosed THEN
			stInOuts.bNozzleStabValve_Q := FALSE;
			iWorkStep := 32;
		ELSIF fbTON.Q THEN
			nQErrorId := nStFix_S06CarrierAndWheelAssyGrease_ErrorCodes.StabilizerReturnTimeout;	
			iWorkStep := 90;
		END_IF
		IF iWorkStep <> 30 THEN fbTON(IN:= FALSE); fbTOF_Delay(IN:= FALSE); END_IF
		
	32:
		fbTON(IN:= TRUE, PT:= T#500MS);
		stInOuts.bRotationStabValve_Q := FALSE;
		IF stInOuts.bRotationStabilizerClosed THEN
			iWorkStep := 34;
		ELSIF fbTON.Q THEN
			nQErrorId := nStFix_S06CarrierAndWheelAssyGrease_ErrorCodes.StabilizerReturnTimeout;
			iWorkStep := 90;
		END_IF
		IF iWorkStep <> 32 THEN fbTON(IN:= FALSE); END_IF
		
	34:	// Kowadło zwolnione
		bQBusy := FALSE;
		bQLocked := FALSE;		
		iWorkStep := 5;
		
	50:	// Manual mode
		bManualWork :=FALSE;
		iWorkStep := 5;
		
	90:		// Błąd w pracy kowadła
		stInOuts.bRotationStabValve_Q := stInOuts.bNozzleStabValve_Q := stInOuts.bGreaseValve_Q := FALSE;
		bQBusy := FALSE;
		bQError := TRUE;
		iWorkStep := 91;
		
	91:
		IF bRelease OR bResetMethod THEN
			bQError := FALSE;
			nQErrorId := iWorkStep := 0;
		END_IF

	ELSE
		mNewEvent(nStFix_S06CarrierAndWheelAssyGrease_ErrorCodes.ProgramConfigError);		
END_CASE

END_FUNCTION_BLOCK

// ProdLineMachines/Sonictech/Fixtures/S06_CarrierWheelLubrification/V2/fbStFix_S06CarrierAndWheelAssyGrease_V2
FUNCTION_BLOCK PUBLIC fbStFix_S06CarrierAndWheelAssyGrease_V2 EXTENDS fbStFixBaseTemplate IMPLEMENTS I_Fixture 
VAR_IN_OUT
	stInOuts:stStFix_S06CarrierAndWheelAssyGrease_V2_InOuts;
END_VAR
VAR_INPUT
	stSettings : stStFix_S06CarrierAndWheelAssyGrease_V2_Settings;
END_VAR
VAR_OUTPUT
END_VAR
VAR
	fbTP_Grease: TP;
	fbBVS :fbBVSControl;
	bErrorBVS : BOOL;
	bWheel : BOOL;
	bGoodSide : BOOL;
	I_Vision: I_VisionSensorSTD;
	iTriggerRepeats: INT;
	iMaxTrigRepeats: INT :=3;
	fbTON_GreaseDelay:TON;
END_VAR

fbTP_Grease(IN:= FALSE, PT:= LIMIT(T#100MS, REAL_TO_TIME(1000*stSettings.rGreaseApplyTime),T#2S), Q=> stInOuts.bGreaseValve_Q);
fbBVS(stIO_Data:=stInOuts.stBvsInOut);
I_Vision := fbBVS;
fbTON_GreaseDelay(IN:= NOT stInOuts.bGreaseValve_Q AND NOT stInOuts.bGreaseSprayValve_Q, PT:= T#200MS);
CASE iWorkStep OF
	0:		// Powrót do stanu początkowego (ustawienie zmiennych)
		bResetMethod := bQReady := bQBusy := bQError := FALSE;
		IF NOT bLock AND NOT bRelease THEN
			fbTON(IN:= FALSE);
			iWorkStep := 1;
		END_IF
			
	1: 		// Sprawdzenie czy siłowniki są w dobrej pozycji itp.
		stInOuts.bRotationStabValve_Q := stInOuts.bNozzleStabValve_Q := stInOuts.bGreaseValve_Q := FALSE;
		bQLocked := FALSE;
		fbTON(IN:= FALSE);
		iWorkStep := 5;
	
	5:		// Oczekiwanie na nowy rozkaz
		bQReady := TRUE;
		bResetMethod:= bReleaseMethod:= bAuxOperMethod:= bLockMethod := FALSE;
		actCheckForNewOrder();
		
	10:		// Blokowanie kowadła
		fbTON(IN:= TRUE, PT:= T#1S);
		stInOuts.bRotationStabValve_Q := TRUE;
		iTriggerRepeats := 0;
		IF stInOuts.bRotationStabilizerClosed THEN
			IF stSettings.bCheckWheelOrientation THEN
				iWorkStep := 11;
			ELSE
				iWorkStep := 13;
			END_IF
		ELSIF fbTON.Q THEN
			mNewEvent(nStFix_S06CarrierAndWheelAssyGrease_V2_ErrorCodes.RotaryFixtureError);		// Brak stabilizacji kowadła w zadanym czasie 135	
		END_IF
		IF iWorkStep <> 10 THEN fbTON(IN:= FALSE); END_IF
  
	11:
		IF I_Vision.mNewInspection(bError => bErrorBVS, bOut1=> bWheel, bOut2=>bGoodSide, bOut3 => ) THEN
			IF 	bErrorBVS THEN // Błąd Czujnika wizyjnego
				nQErrorId := 511;		// Do zmiany	
				iWorkStep := 90;
			END_IF
			
			IF bWheel AND bGoodSide THEN			// Detekcja
				iWorkStep := 13;
			ELSE 
				IF iTriggerRepeats >= iMaxTrigRepeats THEN
					IF bWheel AND NOT bGoodSide THEN
						mNewEvent(nStFix_S06CarrierAndWheelAssyGrease_V2_ErrorCodes.WheelWrongSide);		// Zła strona	
					ELSIF NOT bWheel THEN
						mNewEvent(nStFix_S06CarrierAndWheelAssyGrease_V2_ErrorCodes.LackOfWheel);		// Brak koła	
					ELSE
						mNewEvent(-1);
					END_IF
				ELSE		// Wykonaj powtórne zdjęcie
					iTriggerRepeats := iTriggerRepeats + 1;
					fbTON(IN:= FALSE);
					iWorkStep := 12;
				END_IF
			END_IF
		END_IF
	12: // Oczekiwanie oraz powtórna próba znalezienia
		fbTON(IN:= TRUE, PT:= T#200MS);
		IF fbTON.Q THEN
			fbTON(IN:= FALSE);
			iWorkStep := 11;
		END_IF
		
	13:		// Oczekiwanie na zakończenie detekcji
		fbTON(IN:= TRUE, PT:= T#500MS);
		stInOuts.bNozzleStabValve_Q := TRUE;
		IF stInOuts.bNozzleStabilizerClosed THEN
			iWorkStep := 14;
		ELSIF fbTON.Q THEN
			mNewEvent(nStFix_S06CarrierAndWheelAssyGrease_V2_ErrorCodes.RotaryFixtureError);		// Brak stabilizacji kowadła w zadanym czasie 135	
		END_IF
		IF iWorkStep <> 13 THEN fbTON(IN:= FALSE); END_IF
		
	14:		// Wszystko  OK
		bLock := FALSE;
		bQBusy := FALSE;		
		bQLocked := TRUE;		
		iWorkStep := 5;
		
		
	20: 	// Dodatkowa operacja
		IF bLastOperStatus THEN
			fbTP_Grease(IN:= TRUE);		
			fbTON(IN:= FALSE);	
			iWorkStep := 22;
		ELSE
			bQError := bQBusy := FALSE;	
			bAuxOper := FALSE;
			iWorkStep := 5;
		END_IF
	
	22:	
		IF NOT stInOuts.bGreaseValve_Q THEN
			stInOuts.bGreaseSprayValve_Q := TRUE;
			fbTON(IN:= TRUE, PT:= T#200MS);
			IF fbTON.Q THEN
				stInOuts.bGreaseSprayValve_Q := FALSE;
				bAuxOper := FALSE;
				iWorkStep := 5;
				bQBusy := FALSE;
			END_IF
		END_IF
	
	30:		// Zwalnianie kowadła
		fbTON(IN:= NOT stInOuts.bGreaseValve_Q, PT:= T#2S);
		stInOuts.bNozzleStabValve_Q R= fbTON_GreaseDelay.Q;
		IF stInOuts.bNozzleStabilizerClosed THEN
			iWorkStep := 32;
		ELSIF fbTON.Q THEN
			mNewEvent(-1);
		END_IF
		IF iWorkStep <> 30 THEN fbTON(IN:= FALSE); END_IF
		
	32:
		fbTON(IN:= TRUE, PT:= T#500MS);
		stInOuts.bRotationStabValve_Q := FALSE;
		stInOuts.bNozzleStabValve_Q:= FALSE;
		IF NOT stInOuts.bRotationStabilizerClosed THEN
			iWorkStep := 34;
		ELSIF fbTON.Q THEN
			mNewEvent(-1);
		END_IF
		IF iWorkStep <> 32 THEN fbTON(IN:= FALSE); END_IF
		
	34:	// Kowadło zwolnione
		bRelease := FALSE;
		bQBusy := FALSE;
		bQLocked := FALSE;		
		iWorkStep := 5;
		
	50:		// Manual work coordination
		fbTON(IN:= TRUE, PT:= T#15M);
		IF NOT bManualWork OR fbTON.Q THEN
			fbTON(IN:= FALSE);
			bManualWork := FALSE;
			iWorkStep := 0;
		END_IF
		
	90:		// Błąd w pracy kowadła
		stInOuts.bRotationStabValve_Q := stInOuts.bNozzleStabValve_Q := stInOuts.bGreaseValve_Q := FALSE;
		bQBusy := FALSE;
		bQError := TRUE;
		iWorkStep := 91;
		
	91:
		IF bRelease OR bResetMethod THEN
			bQError := FALSE;
			nQErrorId := iWorkStep := 0;
		END_IF

	ELSE
		mNewEvent(nStFix_S06CarrierAndWheelAssyGrease_V2_ErrorCodes.ProgramConfigError);		
END_CASE

END_FUNCTION_BLOCK

// ProdLineMachines/Sonictech/Fixtures/S07_CarrierAssyWithPiston/V1/fbStFix_S07CarrierPistonAssy
FUNCTION_BLOCK PUBLIC fbStFix_S07CarrierPistonAssy EXTENDS fbStFixBaseTemplate IMPLEMENTS I_Fixture 
VAR_IN_OUT
	stInOuts:stStFix_S07CarrierPistonAssy_InOuts;
END_VAR
VAR_INPUT
	stSettings : stStFix_S07CarrierPistonAssy_Settings;
END_VAR
VAR_OUTPUT
END_VAR
VAR
	uiCtr_Operations:UINT;
	fbTP_Scavenge: TP;
	fbTON_CarrierStabClosed: TON;
END_VAR

fbTP_Scavenge(IN:= FALSE, PT:= REAL_TO_TIME(stSettings.rScavenge_Time_S*1000), Q=> stInOuts.bVacuumScavenge_Q);

CASE iWorkStep OF
	0:		// Powrót do stanu początkowego (ustawienie zmiennych)
		bResetMethod := bQReady := bQBusy := bQError := FALSE;
		IF NOT bLock AND NOT bRelease THEN
			fbTON(IN:= FALSE);
			iWorkStep := 1;
		END_IF
			
	1: 		// Sprawdzenie czy siłowniki są w dobrej pozycji itp.
		stInOuts.bRotationStabValve_Q := stInOuts.bCarierStabValve_Q := stInOuts.bVacuumON_Q := FALSE;
		bQLocked := FALSE;
		fbTON(IN:= FALSE);
		iWorkStep := 5;
	
	5:		// Oczekiwanie na nowy rozkaz
		bQReady := TRUE;
		bResetMethod:= bReleaseMethod:= bAuxOperMethod:= bLockMethod := FALSE;
		stInOuts.bVacuumON_Q := bUserLogged;
		actCheckForNewOrder();
		
	10:		// Blokowanie kowadła
		fbTON(IN:= TRUE, PT:= T#500MS);
		stInOuts.bRotationStabValve_Q := TRUE;
		IF stInOuts.bRotationStabilizerClosed THEN
			fbTON_CarrierStabClosed(IN:= FALSE);
			iWorkStep := 12;
		ELSIF fbTON.Q THEN
			mNewEvent(nStFix_S07CarrierPistonAssy_ErrorCodes.StabilizingTimeout);
		END_IF
		IF iWorkStep <> 10 THEN fbTON(IN:= FALSE); END_IF
  
	12:		// Oczekiwanie na zakończenie blokowania
		fbTON(IN:= TRUE, PT:= T#1S);
		fbTON_CarrierStabClosed(IN:= NOT stInOuts.bCarierStabilizerOpened, PT:= T#200MS);
		stInOuts.bCarierStabValve_Q := TRUE;
		IF fbTON_CarrierStabClosed.Q THEN
			iWorkStep := 14;
		ELSIF fbTON.Q THEN
			mNewEvent(nStFix_S07CarrierPistonAssy_ErrorCodes.StabilizingTimeout);
    	END_IF
		IF iWorkStep <> 12 THEN fbTON(IN:= FALSE); END_IF
		
	14:		// Wszystko  OK
		bQBusy := FALSE;		
		bQLocked := TRUE;		
		iWorkStep := 5;
		
	20: 	// Dodatkowa operacja
		bQError := bQBusy := FALSE;		
		iWorkStep := 5;
		
	30:		// Zwalnianie kowadła
		IF NOT fbTON.IN THEN
			uiCtr_Operations := uiCtr_Operations + 1;
			IF uiCtr_Operations >= stSettings.uiScavengeEveryN AND stSettings.uiScavengeEveryN > 0 THEN
				fbTP_Scavenge(IN:= TRUE);
				uiCtr_Operations := 0;
			END_IF
		END_IF
		fbTON(IN:= TRUE, PT:= T#800MS);
		stInOuts.bCarierStabValve_Q := FALSE;
		IF stInOuts.bCarierStabilizerOpened THEN
			iWorkStep := 32;
		ELSIF fbTON.Q THEN
			mNewEvent(nStFix_S07CarrierPistonAssy_ErrorCodes.StabilizerReturnTimeout);
    	END_IF
		IF iWorkStep <> 30 THEN fbTON(IN:= FALSE); END_IF
		
	32:
		fbTON(IN:= TRUE, PT:= T#800MS);
		stInOuts.bRotationStabValve_Q := FALSE;
		IF NOT stInOuts.bRotationStabilizerClosed THEN
			iWorkStep := 34;
		ELSIF fbTON.Q THEN
			mNewEvent(nStFix_S07CarrierPistonAssy_ErrorCodes.StabilizerReturnTimeout);
		END_IF
		IF iWorkStep <> 32 THEN fbTON(IN:= FALSE); END_IF
		
	34:	// Kowadło zwolnione
		bQBusy := FALSE;
		bQLocked := FALSE;		
		iWorkStep := 5;
		
	50:		// Manual work coordination
		fbTON(IN:= TRUE, PT:= T#15M);
		IF NOT bManualWork OR fbTON.Q THEN
			fbTON(IN:= FALSE);
			bManualWork := FALSE;
			iWorkStep := 0;
		END_IF
		
	90:		// Błąd w pracy kowadła
		stInOuts.bRotationStabValve_Q := stInOuts.bCarierStabValve_Q:= stInOuts.bVacuumScavenge_Q := FALSE;
		bQBusy := FALSE;
		bQError := TRUE;
		iWorkStep := 91;
		
	91:
		IF bRelease OR bResetMethod THEN
			bQError := FALSE;
			nQErrorId := 0;
			iWorkStep := 0;
		END_IF

	ELSE
		mNewEvent(nStFix_S07CarrierPistonAssy_ErrorCodes.ProgramConfigError);		
END_CASE

END_FUNCTION_BLOCK

// ProdLineMachines/Sonictech/Fixtures/S07_CarrierAssyWithPiston/V2/fbStFix_S07CarrierPistonAssy_V2
FUNCTION_BLOCK PUBLIC fbStFix_S07CarrierPistonAssy_V2 EXTENDS fbStFixBaseTemplate IMPLEMENTS I_Fixture 
VAR_IN_OUT
	stInOuts:stStFix_S07CarrierPistonAssy_V2_InOuts;
END_VAR
VAR_INPUT
	// Wejścia cyfrowe, konfiguracyjne itp
	bSafetyGate:BOOL;
	bCarier_OnlyOpenSensor: BOOL:= FALSE;
	stSettings : stStFix_S07CarrierPistonAssy_V2_Settings;
END_VAR
VAR
	uiCtr_Operations:UINT;
	fbTP_Scavenge: TP;
	fbTON_CarrierStabClosed: TON;
	fb_HeatStamp : PID;
	fb_HeatStampPWM: fbPwmGenerator;
	fbPWM: fbPwmGenerator;
	bTurnHeatON: BOOL;
	rHeatStampPower: REAL;
	bUpdatePidParams: BOOL;
	fbHeatStampTempperatureStableFilter: fbBinaryFilter;
	bHeatStampTemperatureStable: BOOL;
	fbHeaterDamage: TON;
	rLastMeasureTemperature : REAL;
	rStampTemperature: REAL;
	bMakeStamp: BOOL;
	iStampWorkStep: INT;
	fbTON_StampTimeout: TON;
	bStampMaked: BOOL;
END_VAR

ACT_HeatStamp();
fbTP_Scavenge(IN:= FALSE, PT:= LIMIT(T#100MS, REAL_TO_TIME(1000*stSettings.rScavenge_Time_S),T#2S), Q=> stInOuts.bVacuumScavenge_Q);

IF bWeldingActive AND stSettings.bHeatStampMakingEnable AND stSettings.bHeatStampMarkWhenWeldingActive AND NOT bStampMaked THEN
	stInOuts.bHeatSafetyGateValve_Q := bMakeStamp := TRUE;
END_IF

CASE iWorkStep OF
	0:		// Powrót do stanu początkowego (ustawienie zmiennych)
		bResetMethod := bQReady := bQBusy := bQError := FALSE;
		IF NOT bLock AND NOT bRelease THEN
			fbTON(IN:= FALSE);
			iWorkStep := 1;
		END_IF
			
	1: 		// Sprawdzenie czy siłowniki są w dobrej pozycji itp.
		stInOuts.bRotationStabValve_Q := stInOuts.bCarierStabValve_Q := stInOuts.bVacuumON_Q := stInOuts.bHeatStampValve_Q := stInOuts.bHeatSafetyGateValve_Q := FALSE;
		bQLocked := FALSE;
		fbTON(IN:= FALSE);
		iWorkStep := 5;
	
	5:		// Oczekiwanie na nowy rozkaz
		bQReady := TRUE;
		bResetMethod:= bReleaseMethod:= bAuxOperMethod:= bLockMethod := FALSE;
		stInOuts.bVacuumON_Q := bUserLogged;
		actCheckForNewOrder();
		
	10:		// Blokowanie kowadła
		IF (bHeatStampTemperatureStable AND stSettings.bHeatStampMakingEnable) OR NOT stSettings.bHeatStampMakingEnable THEN 					//Sprawdzenie czy temperatura stempla jest stabilna (mieści się w zadeklarowanej toleracji)
			fbTON(IN:= TRUE, PT:= T#500MS);
			stInOuts.bRotationStabValve_Q := TRUE;
			IF stInOuts.bRotationStabilizerClosed AND stInOuts.bCarierStabilizerOpened THEN
				fbTON_CarrierStabClosed(IN:= FALSE);
				iWorkStep := 12;
			ELSIF fbTON.Q THEN
				mNewEvent(nStFix_S07CarrierPistonAssy_V2_ErrorCodes.RotaryFixtureError);		// Brak stabilizacji kowadła w zadanym czasie 135	
			END_IF		
		ELSE
			mNewEvent(nStFix_S07CarrierPistonAssy_V2_ErrorCodes.HeatStampTempStabWait);			// numer błędu do zmiany	
		END_IF
		IF iWorkStep <> 10 THEN fbTON(IN:= FALSE); END_IF
  
	12:		// Oczekiwanie na zakończenie blokowania
		fbTON(IN:= TRUE, PT:= T#1S);
		IF bCarier_OnlyOpenSensor THEN
			fbTON_CarrierStabClosed(IN:= NOT stInOuts.bCarierStabilizerOpened, PT:= T#400MS);
		ELSE
			fbTON_CarrierStabClosed.IN S=stInOuts.bCarierStabilizerClosed;
			fbTON_CarrierStabClosed(PT:= T#100MS);
		END_IF
		stInOuts.bCarierStabValve_Q := TRUE;
		IF fbTON_CarrierStabClosed.Q THEN
			iWorkStep := 14;
		ELSIF fbTON.Q THEN
			mNewEvent(nStFix_S07CarrierPistonAssy_V2_ErrorCodes.CylinderFixtureError);		// Brak stabilizacji kowadła w zadanym czasie 135	
		END_IF
		IF iWorkStep <> 12 THEN fbTON(IN:= FALSE); END_IF
		
	14:		// Wszystko  OK
		bLock := bQBusy := FALSE;		
		bQLocked := TRUE;		
		iWorkStep := 5;
		
		
	20: 	// Operacja wykonana - trzeba wykonać przedmuch?
		uiCtr_Operations := uiCtr_Operations + 1;
		IF uiCtr_Operations>= stSettings.uiScavengeEveryN AND stSettings.uiScavengeEveryN > 0 THEN
			fbTP_Scavenge(IN:= TRUE);
			uiCtr_Operations := 0;
		END_IF
		stInOuts.bHeatSafetyGateValve_Q := bMakeStamp := stSettings.bHeatStampMakingEnable AND bLastOperStatus AND NOT stSettings.bHeatStampMarkWhenWeldingActive;
		iWorkStep := 21;
		
	21:	
		bAuxOper := bQError := bQBusy := FALSE;		
		iWorkStep := 5;
		
		
	30:		// Zwalnianie kowadła
		fbTON(IN:= TRUE, PT:= T#800MS);
		stInOuts.bCarierStabValve_Q := FALSE;
		IF stInOuts.bCarierStabilizerOpened THEN
			iWorkStep := 32;
		ELSIF fbTON.Q THEN
			mNewEvent(nStFix_S07CarrierPistonAssy_V2_ErrorCodes.CylinderFixtureError);		// Brak stabilizacji kowadła w zadanym czasie 135	
		END_IF
		IF iWorkStep <> 30 THEN fbTON(IN:= FALSE); END_IF
		
	32:
		fbTON(IN:= TRUE, PT:= T#800MS);
		stInOuts.bRotationStabValve_Q := FALSE;
		IF NOT stInOuts.bRotationStabilizerClosed THEN
			iWorkStep := 34;
		ELSIF fbTON.Q THEN
			mNewEvent(nStFix_S07CarrierPistonAssy_V2_ErrorCodes.RotaryFixtureError);		// Brak stabilizacji kowadła w zadanym czasie 135	
		END_IF
		IF iWorkStep <> 32 THEN fbTON(IN:= FALSE); END_IF
		
	34:	// Oczekiwanie na brak znakowania
		IF NOT bMakeStamp OR NOT stSettings.bHeatStampMakingEnable THEN
			iWorkStep := 36;
		END_IF
	
	36:	// Kowadło zwolnione
		bRelease:= bQBusy := FALSE;
		bQLocked := FALSE;		
		iWorkStep := 5;

	50:		// Manual work coordination
		fbTON(IN:= TRUE, PT:= T#15M);
		IF NOT bManualWork OR fbTON.Q THEN
			fbTON(IN:= FALSE);
			bManualWork := FALSE;
			iWorkStep := 0;
		END_IF
		
	90:		// Błąd w pracy kowadła
		stInOuts.bRotationStabValve_Q := stInOuts.bCarierStabValve_Q:= stInOuts.bVacuumScavenge_Q := stInOuts.bHeatStampValve_Q := FALSE;
		stInOuts.bHeatSafetyGateValve_Q R= stInOuts.bHeatStampClosed;
		bQBusy := FALSE;
		bQError := TRUE;
		iWorkStep := 91;
		
	91:
		IF bRelease OR bResetMethod THEN
			iStampWorkStep := 0;
			bMakeStamp := FALSE;
			stInOuts.bHeatSafetyGateValve_Q R= stInOuts.bHeatStampClosed;
			bQError := FALSE;
			nQErrorId := 0;
			iWorkStep := 0;
		END_IF
		
	ELSE
		mNewEvent(nStFix_S07CarrierPistonAssy_V2_ErrorCodes.ProgramConfigError);
END_CASE

ACTION ACT_HeatStamp:
rStampTemperature := INT_TO_REAL(stInOuts.rHeatStampTemperature)/10; // Przepisanie temperatury
fb_HeatStamp(	// Regulacja temperatury grzałki
	ACTUAL:= rStampTemperature, 
	SET_POINT:= stSettings.rHeatStampSetTemperature, 
	KP:= 3.9,	//stSettings.rHeatStamp_Kp, 
	TN:= 39,	//stSettings.rHeatStamp_Ki, 
	TV:= 0,		//stSettings.rHeatStamp_Kd, 
	Y_MANUAL:= 30.0, 
	Y_OFFSET:= , 
	Y_MIN:= 00.0, 
	Y_MAX:= 95.0, 
	MANUAL:= NOT stSettings.bHeatStampMakingEnable OR stInOuts.bAI_StampTemperature_Error, 
	RESET:= bUpdatePidParams, 
	Y=> rHeatStampPower);
	bUpdatePidParams:=FALSE;
//Sygnał PWM dla SSR
fbPWM(bEnable := stSettings.bHeatStampMakingEnable, rCycleInS := 0.5, rDutyCyclePercent:= rHeatStampPower, bOutput => stInOuts.bHeatStampPWMSignal);

fbHeatStampTempperatureStableFilter(IN:= ABS(stSettings.rHeatStampSetTemperature - rStampTemperature) <= stSettings.rHeatStampAllowDeviation, 
									 tON:= T#30S, tOFF := T#5S, Q => bHeatStampTemperatureStable);

fbHeaterDamage(IN:=stSettings.bHeatStampMakingEnable AND fbHeaterDamage.Q, PT:= T#5S);
(*IF fbHeaterDamage.Q THEN
	IF ABS(rStampTemperature - rLastMeasureTemperature) < 0.2 AND NOT bHeatStampTemperatureStable AND   THEN
		nQErrorId := nStFix_S07CarrierPistonAssy_V2_ErrorCodes.DamagedStamp;		// Grzałka bądź termopara uszkodzona	
		iWorkStep := 90;
	END_IF
	rLastMeasureTemperature := rStampTemperature;
END_IF	*)


CASE iStampWorkStep OF 
	0:	// Oczekiwanie na znakowanie
		IF bMakeStamp THEN
			bStampMaked := FALSE;
			IF bHeatStampTemperatureStable THEN 					//Sprawdzenie czy temperatura stempla jest stabilna (mieści się w zadeklarowanej toleracji)
				fbTON_StampTimeout(IN:= FALSE);
				iStampWorkStep := 5;
			ELSE
				mNewEvent(nStFix_S07CarrierPistonAssy_V2_ErrorCodes.HeatStampTempStabWait);
			END_IF	
		END_IF
		
	5:	// Otwarcie bramki
		fbTON_StampTimeout(IN:= TRUE, PT:= T#1S);
		stInOuts.bHeatSafetyGateValve_Q := TRUE;
		IF stInOuts.bStampSafetyGateOpened OR NOT bSafetyGate THEN
			iStampWorkStep := 10;
		ELSIF fbTON_StampTimeout.Q THEN
			mNewEvent(nStFix_S07CarrierPistonAssy_V2_ErrorCodes.HeatStampTempStabWait);
		END_IF
		IF iStampWorkStep <> 5 THEN fbTON_StampTimeout(IN:= FALSE); END_IF

	10:	// Znakowanie - oczekiwanie na otwarcie 		
		fbTON_StampTimeout(IN:= TRUE, PT:= T#1S);
		stInOuts.bHeatStampValve_Q := TRUE;
		IF stInOuts.bHeatStampOpened THEN
			iStampWorkStep := 15;
		ELSIF fbTON_StampTimeout.Q THEN
			mNewEvent(nStFix_S07CarrierPistonAssy_V2_ErrorCodes.HeatStampWorkError);
		END_IF
		IF iStampWorkStep <> 10 THEN fbTON_StampTimeout(IN:= FALSE); END_IF
		
	15:	// Znakowanie przez pewien czas
		fbTON_StampTimeout(IN:= TRUE, PT:= LIMIT(T#100MS,REAL_TO_TIME(1000*stSettings.rHeatStampMarkingTime),T#2S));
		IF fbTON_StampTimeout.Q  THEN
			stInOuts.bHeatStampValve_Q := FALSE;
			iStampWorkStep := 20;
		END_IF
		
	20:	// Powrót siłownika
		fbTON_StampTimeout(IN:= TRUE, PT:= T#1S);
		stInOuts.bHeatStampValve_Q := FALSE;
		IF stInOuts.bHeatStampClosed THEN
			stInOuts.bHeatSafetyGateValve_Q := FALSE;
			iStampWorkStep := 25;
		ELSIF fbTON_StampTimeout.Q THEN
			mNewEvent(nStFix_S07CarrierPistonAssy_V2_ErrorCodes.HeatStampWorkError);
		END_IF
		IF iStampWorkStep <> 20 THEN fbTON_StampTimeout(IN:= FALSE); END_IF
		
	25:	// Oczekiwanie na zamknięcie bramki
		fbTON_StampTimeout(IN:= TRUE, PT:= T#1S);
		stInOuts.bHeatSafetyGateValve_Q := FALSE;
		IF NOT stInOuts.bStampSafetyGateOpened OR NOT bSafetyGate THEN
			iStampWorkStep := 0;
			bMakeStamp := FALSE;	
			bStampMaked := TRUE;
		ELSIF fbTON_StampTimeout.Q THEN
			mNewEvent(nStFix_S07CarrierPistonAssy_V2_ErrorCodes.HeatStampWorkError);
		END_IF
		IF iStampWorkStep <> 25 THEN fbTON_StampTimeout(IN:= FALSE); END_IF
END_CASE
END_ACTION

METHOD PROTECTED mNewEvent
VAR_INPUT
	nErrID: INT;
END_VAR
bQError := TRUE;
nQErrorId := nErrID;
iWorkStep := 90;
iStampWorkStep := 0;
bMakeStamp := FALSE;
END_METHOD

END_FUNCTION_BLOCK

// ProdLineMachines/Sonictech/Fixtures/S08_CoolerClosure/V1/fbStFix_S08CoolerClosure
FUNCTION_BLOCK PUBLIC fbStFix_S08CoolerClosure EXTENDS fbStFixBaseTemplate IMPLEMENTS I_Fixture
VAR_IN_OUT
	stInOuts:stStFix_S08CoolerClosure_InOuts;
END_VAR
VAR
	fbTON_CarrierStabClosed: TON;
END_VAR


CASE iWorkStep OF
	0:		// Powrót do stanu początkowego (ustawienie zmiennych)
		bResetMethod := bQReady := bQBusy := bQError := FALSE;
		IF NOT bLock AND NOT bRelease THEN
			fbTON(IN:= FALSE);
			iWorkStep := 1;
		END_IF
			
	1: 		// Sprawdzenie czy siłowniki są w dobrej pozycji itp.
		stInOuts.bRotationStabValve_Q:= FALSE;
		bQLocked := FALSE;
		fbTON(IN:= FALSE);
		iWorkStep := 5;
	
	5:		// Oczekiwanie na nowy rozkaz
		bQReady := TRUE;
		bResetMethod:= bReleaseMethod:= bAuxOperMethod:= bLockMethod := FALSE;
		actCheckForNewOrder();
		
	10:		// Blokowanie kowadła
		fbTON(IN:= TRUE, PT:= T#1S);
		stInOuts.bRotationStabValve_Q := TRUE;
		IF stInOuts.bRotationStabilizerClosed THEN
			iWorkStep := 12;
		ELSIF fbTON.Q THEN
			mNewEvent(nStFix_S08CoolerClosure_ErrorCodes.PartStabilizationTimeout);
		END_IF
		IF iWorkStep <> 10 THEN fbTON(IN:= FALSE); END_IF
  		
	12:		// Wszystko  OK
		bQBusy := FALSE;		
		bQLocked := TRUE;		
		iWorkStep := 5;
		
	20: 	// Dodatkowa operacja
		bQError := bQBusy := FALSE;		
		iWorkStep := 5;
		
	30:		// Zwalnianie kowadła
		fbTON(IN:= TRUE, PT:= T#2S);
		stInOuts.bRotationStabValve_Q := FALSE;
		IF NOT stInOuts.bRotationStabilizerClosed THEN
			iWorkStep := 32;
		ELSIF fbTON.Q THEN
			mNewEvent(nStFix_S08CoolerClosure_ErrorCodes.PartStabReleaseTimeout);
		END_IF
		IF iWorkStep <> 30 THEN fbTON(IN:= FALSE); END_IF
			
	32:	// Kowadło zwolnione
		bQBusy := FALSE;
		bQLocked := FALSE;		
		iWorkStep := 5;
		
	90:		// Błąd w pracy kowadła
		stInOuts.bRotationStabValve_Q := FALSE;
		bQBusy := FALSE;
		bQError := TRUE;
		iWorkStep := 91;
		
	91:
		IF bRelease OR bResetMethod THEN
			bQError := FALSE;
			nQErrorId := 0;
			iWorkStep := 0;
		END_IF
		
END_CASE

END_FUNCTION_BLOCK

// ProdLineMachines/Sonictech/Fixtures/S08_CoolerClosure/V2/fbStFix_S08CoolerClosure_V2
FUNCTION_BLOCK PUBLIC fbStFix_S08CoolerClosure_V2 EXTENDS fbStFixBaseTemplate IMPLEMENTS I_Fixture
VAR_IN_OUT
	stInOuts:stStFix_S08CoolerClosure_V2_InOuts;
END_VAR
VAR_INPUT
	iMaxTrigRepeats: INT :=1;
	stSettings : stStFix_S08CoolerClosure_V2_Settings;
END_VAR
VAR_OUTPUT
END_VAR
VAR
	fbTONWaitForReset: TON;
	bErrorBVS : BOOL;
	bStamp : BOOL;
	bPosition: BOOL;
	bPartInside: BOOL;
	fbBVS :fbBVSControl;
	I_Vision: I_VisionSensorSTD;
	iTriggerRepeats: INT;
	fbTONRelease: TON;
END_VAR

fbBVS(stIO_Data:=stInOuts.stBvsInOut);
I_Vision := fbBVS;


CASE iWorkStep OF
	0:		// Powrót do stanu początkowego (ustawienie zmiennych)
		fbTONWaitForReset(IN:=TRUE,PT:=T#350MS);
		IF fbTONWaitForReset.Q THEN
			stInOuts.bBiggerStabilizerClose := stInOuts.bSmallerStabilizerClose :=  FALSE;
		END_IF
		bResetMethod := bQReady := bQBusy := bQError := FALSE;
		IF NOT stInOuts.bBiggerStabilizerClose AND NOT stInOuts.bSmallerStabilizerClose THEN
			stInOuts.bCarierUpPosition := FALSE;
			fbTONWaitForReset(IN:=FALSE);
			iWorkStep := 1;
		END_IF
		IF iWorkStep <> 1 THEN fbTON(IN:= FALSE); END_IF
		
	1: 		// Sprawdzenie czy siłowniki są w dobrej pozycji itp.
		bQLocked := FALSE;
		fbTON(IN:= FALSE);
		iWorkStep := 5;
		IF iWorkStep <> 1 THEN fbTON(IN:= FALSE); END_IF
		
	5:		// Oczekiwanie na nowy rozkaz
		IF NOT bQLocked THEN
			stInOuts.bCarierClose := FALSE;
		END_IF
		bQReady := TRUE;
		bResetMethod:= bReleaseMethod:= bAuxOperMethod:= bLockMethod := FALSE;
		actCheckForNewOrder();
		
	10:	// 
		IF stSettings.bCheckVisionSign THEN
			iWorkStep := 11;
		ELSE
			iWorkStep := 14;
		END_IF
			
	11:	// Sprawdzenie Vision
		IF I_Vision.mNewInspection(bError => bErrorBVS, bOut1=>bPosition , bOut2=>bPartInside, bOut3 =>bStamp ) THEN
			IF 	bErrorBVS THEN // Błąd Czujnika wizyjnego
				mNewEvent(nStFix_S08CoolerClosure_V2_ErrorCodes.VisionSensorError);
			END_IF	
			IF bStamp AND bPosition AND bPartInside  THEN			// Detekcja
				iWorkStep := 14;
				iTriggerRepeats:= 0;
			ELSE 
				IF iTriggerRepeats >= iMaxTrigRepeats THEN
					IF NOT bStamp THEN
						mNewEvent(nStFix_S08CoolerClosure_V2_ErrorCodes.HeatStampNotDetected);	
					END_IF
				ELSE		// Wykonaj powtórne zdjęcie
					iTriggerRepeats := iTriggerRepeats + 1;
					fbTON(IN:= FALSE);
					iWorkStep := 12;
				END_IF
			END_IF
		END_IF
		
	12: // Oczekiwanie oraz powtórna próba znalezienia
		fbTON(IN:= TRUE, PT:= T#200MS);
		IF fbTON.Q THEN
			fbTON(IN:= FALSE);
			iWorkStep := 11;
		END_IF
		
		
	14:		// Blokowanie kowadła
		fbTON(IN:= TRUE, PT:= T#2S);
		IF stSettings.bBiggerActuatorFirst THEN
			stInOuts.bBiggerStabilizerClose := TRUE;
			stInOuts.bSmallerStabilizerClose S= stInOuts.bBiggerStabilizerClosed AND stInOuts.bCarierUpPosition; 
		ELSE
			stInOuts.bSmallerStabilizerClose := TRUE;
			stInOuts.bBiggerStabilizerClose S= stInOuts.bSmallerStabilizerClosed AND stInOuts.bCarierUpPosition;
		END_IF
		stInOuts.bCarierClose S= stInOuts.bBiggerStabilizerClosed AND stInOuts.bSmallerStabilizerClosed AND stInOuts.bCarierUpPosition;
		IF stInOuts.bBiggerStabilizerClosed AND stInOuts.bSmallerStabilizerClosed AND NOT stInOuts.bCarierUpPosition THEN
			iWorkStep := 16;
		END_IF		
		IF fbTON.Q THEN
			IF stInOuts.bSmallerStabilizerClose AND NOT stInOuts.bSmallerStabilizerClosed THEN
				mNewEvent(nStFix_S08CoolerClosure_V2_ErrorCodes.SmallerActuatorError);
			ELSIF stInOuts.bBiggerStabilizerClose AND NOT stInOuts.bBiggerStabilizerClosed THEN
				mNewEvent(nStFix_S08CoolerClosure_V2_ErrorCodes.BiggerActuatorError);
			ELSIF stInOuts.bCarierClose AND stInOuts.bCarierUpPosition THEN
				mNewEvent(nStFix_S08CoolerClosure_V2_ErrorCodes.CoolerActuatorError);
			END_IF
		END_IF
		IF iWorkStep <> 14 THEN fbTON(IN:= FALSE); END_IF

	16:		// Wszystko  OK
		bQBusy := FALSE;		
		bQLocked := TRUE;		
		iWorkStep := 5;
		
	20: 	// Dodatkowa operacja
		bQError := bQBusy := FALSE;		
		iWorkStep := 5;
	
	30:		// Zwalnianie kowadła
		fbTON(IN:= TRUE, PT:= T#2S);
		fbTONRelease(IN:=TRUE,PT:=T#350MS);
		
		stInOuts.bSmallerStabilizerClose := FALSE; //R= fbTONRelease.Q;
		stInOuts.bBiggerStabilizerClose R= stInOuts.bSmallerStabilizerOpened;
		stInOuts.bCarierClose R= stInOuts.bBiggerStabilizerOpened AND stInOuts.bSmallerStabilizerOpened;
		IF stInOuts.bSmallerStabilizerOpened AND stInOuts.bBiggerStabilizerOpened AND stInOuts.bCarierUpPosition THEN
			iWorkStep := 32;
		END_IF
		IF fbTON.Q THEN
			IF NOT stInOuts.bSmallerStabilizerClose AND stInOuts.bSmallerStabilizerClosed THEN
				mNewEvent(nStFix_S08CoolerClosure_V2_ErrorCodes.SmallerActuatorError);
			ELSIF NOT stInOuts.bBiggerStabilizerClose AND stInOuts.bBiggerStabilizerClosed THEN
				mNewEvent(nStFix_S08CoolerClosure_V2_ErrorCodes.BiggerActuatorError);
			ELSIF stInOuts.bCarierClose AND stInOuts.bCarierUpPosition THEN
				mNewEvent(nStFix_S08CoolerClosure_V2_ErrorCodes.CoolerActuatorError);
			END_IF
		END_IF
		IF iWorkStep <> 30 THEN fbTON(IN:= FALSE);fbTONRelease(IN:=FALSE); END_IF
			
	32:	// Kowadło zwolnione
		bQBusy := FALSE;
		bQLocked := FALSE;		
		iWorkStep := 5;
		stInOuts.bCarierClose := FALSE;

	50:		// Manual work coordination
		fbTON(IN:= TRUE, PT:= T#15M);
		IF NOT bManualWork OR fbTON.Q THEN
			fbTON(IN:= FALSE);
			bManualWork := FALSE;
			iWorkStep := 0;
		END_IF
		
	90:		// Błąd w pracy kowadła
		bQBusy := FALSE;
		bQError := TRUE;
		iWorkStep := 91;
		
	91:
		IF bRelease OR bResetMethod THEN
			bQError := FALSE;
			nQErrorId := iWorkStep := 0;
			stInOuts.bCarierClose:=FALSE;
		END_IF

	ELSE
		mNewEvent(nStFix_S08CoolerClosure_V2_ErrorCodes.ProgramConfigError);
END_CASE

END_FUNCTION_BLOCK

// ProdLineMachines/Sonictech/Fixtures/S10_CoolerCarrierOrifice/fbStFix_S10CoolerCarrierOrifice
FUNCTION_BLOCK PUBLIC fbStFix_S10CoolerCarrierOrifice EXTENDS fbStFixBaseTemplate IMPLEMENTS I_Fixture 
VAR_IN_OUT
	stInOuts:stStFix_S10CoolerCarrierOrifice_InOuts;
END_VAR
VAR_INPUT
END_VAR
VAR_OUTPUT
END_VAR
VAR
	fbTON_ROtStabOpenDelay: TON;
END_VAR


CASE iWorkStep OF
	0:		// Powrót do stanu początkowego (ustawienie zmiennych)
		bResetMethod := bQReady := bQBusy := bQError := FALSE;
		IF NOT bLock AND NOT bRelease THEN
			fbTON(IN:= FALSE);
			iWorkStep := 1;
		END_IF
			
	1: 		// Sprawdzenie czy siłowniki są w dobrej pozycji itp.
		stInOuts.bRotationStabValve_Q := stInOuts.bStabLockValve_Q := FALSE;
		bQLocked := FALSE;
		fbTON(IN:= FALSE);
		iWorkStep := 5;
	
	5:		// Oczekiwanie na nowy rozkaz
		bQReady := TRUE;
		bResetMethod:= bReleaseMethod:= bAuxOperMethod:= bLockMethod := FALSE;
		actCheckForNewOrder();
		
	10:		// Blokowanie kowadła
		fbTON(IN:= TRUE, PT:= T#2S);
		stInOuts.bRotationStabValve_Q := TRUE;
		IF stInOuts.bRotationStabilizerClosed THEN
			iWorkStep := 14;
		ELSIF fbTON.Q THEN
			nQErrorId := 0;		// Brak stabilizacji kowadła w zadanym czasie 135	
			iWorkStep := 90;
		END_IF
		IF iWorkStep <> 10 THEN fbTON(IN:= FALSE); END_IF
  
(*	12:		// Oczekiwanie na zakończenie detekcji
		fbTON(IN:= TRUE, PT:= T#1S);
		stInOuts.bStabLockValve_Q := TRUE;
		IF stInOuts.bStabilizerLockClosed THEN
			iWorkStep := 14;
		ELSIF fbTON.Q THEN
			nQErrorId := 0;		// Brak stabilizacji kowadła w zadanym czasie 135	
			iWorkStep := 90;
		END_IF
		IF iWorkStep <> 12 THEN fbTON(IN:= FALSE); END_IF
		*)
		
	14:		// Wszystko  OK
		bQBusy := FALSE;		
		bQLocked := TRUE;		
		iWorkStep := 5;
		
	20: 	// Dodatkowa operacja
		bQError := bQBusy := FALSE;		
		iWorkStep := 5;
		
	(*30:		// Zwalnianie kowadła
		fbTON(IN:= TRUE, PT:= T#1S);
		stInOuts.bStabLockValve_Q := FALSE;
		fbTON_ROtStabOpenDelay(IN:= NOT stInOuts.bStabilizerLockClosed, PT:= T#200MS);
		IF fbTON_ROtStabOpenDelay.Q THEN
			iWorkStep := 32;
		ELSIF fbTON.Q THEN
			nQErrorId := 0;		// Brak stabilizacji kowadła w zadanym czasie 135	
			iWorkStep := 90;
		END_IF
		IF iWorkStep <> 30 THEN fbTON(IN:= FALSE); END_IF*)
		
	30: // To był krok 32 - zmiana dla kowadła z 1 siłownikiem
		fbTON(IN:= TRUE, PT:= T#1S);
		stInOuts.bRotationStabValve_Q := FALSE;
		IF NOT stInOuts.bRotationStabilizerClosed THEN
			iWorkStep := 34;
		ELSIF fbTON.Q THEN
			nQErrorId := 0;		// Brak stabilizacji kowadła w zadanym czasie 135	
			iWorkStep := 90;
		END_IF
		IF iWorkStep <> 32 THEN fbTON(IN:= FALSE); END_IF
		
	34:	// Kowadło zwolnione
		bQBusy := FALSE;
		bQLocked := FALSE;		
		iWorkStep := 5;
		
	50:		// Manual work coordination
		fbTON(IN:= TRUE, PT:= T#15M);
		IF NOT bManualWork OR fbTON.Q THEN
			fbTON(IN:= FALSE);
			bManualWork := FALSE;
			iWorkStep := 0;
		END_IF
		
	90:		// Błąd w pracy kowadła
		stInOuts.bRotationStabValve_Q := stInOuts.bStabLockValve_Q := FALSE;
		bQBusy := FALSE;
		bQError := TRUE;
		iWorkStep := 91;
		
	91:
		IF bRelease OR bResetMethod THEN
			bQError := FALSE;
			nQErrorId := 0;
			iWorkStep := 0;
		END_IF

	ELSE
		mNewEvent(-1);	
END_CASE

END_FUNCTION_BLOCK

// ProdLineMachines/Sonictech/Fixtures/S16_FixAndFrontFanDetection/fbStFix_S16PinWeldFfDetection
FUNCTION_BLOCK PUBLIC fbStFix_S16PinWeldFfDetection EXTENDS fbStFixBaseTemplate IMPLEMENTS I_Fixture 
VAR_IN_OUT
	stInOuts:stStFix_S16PinWeldFfDetection_InOuts;
END_VAR
VAR_INPUT
	tSensorFilterTime:TIME:= T#200MS;
	stTestParams:stStFix_S16PinWeldFfDetection_Settings;
	bEnclosureSensInvert	: BOOL;
	iMaxTrigRepeats: INT := 3;

END_VAR
VAR_OUTPUT
	
END_VAR
VAR
	fbBVS: fbBvsControl;
	I_Vision: I_VisionSensorSTD;
	fbEnclosureSensorFilter: fbBinaryFilter;
	iTriggerRepeats: INT;
	bErrorBVS: BOOL;
	
	bSearchAreaVisible: BOOL;
	bFrontFanDetected: BOOL;
	bPartInFixture: BOOL;
	bPartWelded: BOOL;
	iCtr_SensorWorkVerification: INT;	// Value reset at every part pull up from fixture
END_VAR

fbBVS( stIO_Data:= stInOuts.stBalluff, tMinImpWidth:= T#30MS);
I_Vision := fbBVS;

fbEnclosureSensorFilter(IN := stInOuts.bEnclosureSensor XOR bEnclosureSensInvert, tON := tSensorFilterTime, tOFF := tSensorFilterTime/2);
bPartInFixture S= fbEnclosureSensorFilter.RTrig;

IF fbEnclosureSensorFilter.FTrig THEN	// Wyjęcie części z kowadła
	IF stTestParams.NoWeldLockCheck AND bPartInFixture AND NOT bPartWelded THEN
		nQErrorId := nStFix_S16PinWeldFfDetection_ErrorCodes.PartsNotWelded;
		iWorkStep := 90;
	END_IF
	bPartInFixture := bPartWelded := FALSE;
	iCtr_SensorWorkVerification := 0;
END_IF

CASE iWorkStep OF
	0:		// Powrót do stanu początkowego (ustawienie zmiennych)
		bResetMethod := bQReady := bQBusy := bQError := FALSE;
		stInOuts.bEnclosureLock_Q := stInOuts.bRotationStabValve_Q := FALSE;
		fbBVS.bTrigger := FALSE;
		IF NOT bLock AND NOT bRelease THEN
			fbTON(IN:= FALSE);
			iWorkStep := 1;
		END_IF
			
	1: 		// Sprawdzenie czy siłowniki są w dobrej pozycji itp.
		bQLocked := FALSE;
		iWorkStep := 5;
	
	5:		// Oczekiwanie na nowy rozkaz
		stInOuts.bEnclosureLock_Q S= bUserLogged AND fbEnclosureSensorFilter.RTrig;
		bResetMethod:= bReleaseMethod:= bAuxOperMethod:= bLockMethod := FALSE;
		bQReady := TRUE;
		actCheckForNewOrder();
		
	10:		// Blokowanie kowadła
		IF NOT fbEnclosureSensorFilter.Q AND stTestParams.NoWeldLockCheck THEN
			nQErrorId := nStFix_S16PinWeldFfDetection_ErrorCodes.PartNotDetectedInFixture;		
			iWorkStep := 90;
		ELSIF iCtr_SensorWorkVerification > 2 AND stTestParams.NoWeldLockCheck THEN
			nQErrorId := nStFix_S16PinWeldFfDetection_ErrorCodes.SensorWorkError;		
			iWorkStep := 90;
		ELSE
			nQErrorId := iTriggerRepeats := 0;
//			stInOuts.bRotationStabValve_Q := TRUE;
			IF stTestParams.bFrontFanCheckEN THEN
				iWorkStep := 12;
			ELSE
				iWorkStep := 16;	
			END_IF
		END_IF
		
	12:		// Oczekiwanie na zakończenie detekcji
		IF I_Vision.mNewInspection(bError => bErrorBVS, bOut1=> bSearchAreaVisible, bOut2=>bFrontFanDetected, bOut3 => ) THEN
			IF NOT bErrorBVS THEN		// Balluff odpowiedział
				IF (bSearchAreaVisible OR NOT stTestParams.bIsSearchAreaVisibleCheckEN) AND bFrontFanDetected THEN		// Wszystko wykryte
					iWorkStep := 16;
				ELSE		// NIe wyszystko wykryte
					IF iTriggerRepeats >= iMaxTrigRepeats THEN		// Wykonano powtórne zdjęcie
						IF NOT bSearchAreaVisible AND stTestParams.bIsSearchAreaVisibleCheckEN THEN
							nQErrorId := nStFix_S16PinWeldFfDetection_ErrorCodes.SearchAreaNotVisible;
						ELSE
							nQErrorId := nStFix_S16PinWeldFfDetection_ErrorCodes.FrontFanNotDetected;
						END_IF
						iWorkStep := 90;
					ELSE		// Wykonaj powtórne zdjęcie
						iTriggerRepeats := iTriggerRepeats + 1;
						fbTON(IN:= FALSE);
						iWorkStep := 14;
					END_IF
				END_IF
			ELSE		// brak odpowiedzi Balluffa
				nQErrorId := nStFix_S16PinWeldFfDetection_ErrorCodes.SensorNotReady;
				iWorkStep := 90;
			END_IF
		END_IF
		
	14:		// Oczekiwanie oraz powtórna próba znalezienia
		fbTON(IN:= TRUE, PT:= T#200MS);
		IF fbTON.Q THEN
			fbTON(IN:= FALSE);
			iWorkStep := 12;
		END_IF
		
	16:		// Wszystko wykryte OK, zablokuj część
		fbTON(IN:= TRUE, PT:= T#500MS);
		stInOuts.bRotationStabValve_Q := TRUE;
		IF fbTON.Q OR stInOuts.bRotationStabilizerClosed THEN
			fbTON(IN:= FALSE);
			bQError := bQBusy := FALSE;
			bQLocked := TRUE;
			iWorkStep := 5;
		END_IF
		
	20:		// Dodatkowa operacja	
		bPartWelded:= TRUE;
		IF stTestParams.NoWeldLockCheck THEN
			iCtr_SensorWorkVerification := iCtr_SensorWorkVerification + 1;	
		END_IF
		bQBusy := FALSE;
		iWorkStep := 5;
	
	30:		// Zwalnianie kowadła
		fbTON(IN:= TRUE, PT:= T#500MS);
		stInOuts.bRotationStabValve_Q := FALSE;
		IF fbTON.Q THEN //OR NOT stInOuts.bRotationStabilizerClosed THEN
			fbTON(IN:= FALSE);
			stInOuts.bEnclosureLock_Q := FALSE;
			iWorkStep := 32;
		END_IF	

	32:	// Kowadło zwolnione
		bQBusy := FALSE;
		bQLocked := FALSE;		
		iWorkStep := 5;
		
	50:		// Manual work coordination
		fbTON(IN:= TRUE, PT:= T#15M);
		IF NOT bManualWork OR fbTON.Q THEN
			fbTON(IN:= FALSE);
			bManualWork := FALSE;
			iWorkStep := 0;
		END_IF
		
	90:		// Błąd w pracy kowadła
		bQBusy := FALSE;
		bQError := TRUE;
		fbBVS.bTrigger := fbBVS.bReadActualInspection := fbBVS.bChangeInspection := FALSE;
		iWorkStep := 91;
		
	91:
		IF bRelease OR bResetMethod THEN
			bQError := FALSE;
			stInOuts.bEnclosureLock_Q := stInOuts.bRotationStabValve_Q := FALSE;
			bQLocked := FALSE;
			nQErrorId := 0;
			iWorkStep := 0;
		END_IF
		
	ELSE
		mNewEvent(nStFix_S16PinWeldFfDetection_ErrorCodes.ProgramConfigError);		
END_CASE

END_FUNCTION_BLOCK

// ProdLineMachines/Sonictech/Fixtures/S17_EnclosurePressFix/fbStFix_S17EnclosureWelding
FUNCTION_BLOCK PUBLIC fbStFix_S17EnclosureWelding EXTENDS fbStFixBaseTemplate IMPLEMENTS I_Fixture 
VAR_IN_OUT
	stInOuts : stStFix_S17EnclosureWelding_InOuts;
END_VAR
VAR_INPUT
	tSensorFilterTime:TIME:= T#200MS;
	bEnclosureSensorInvert:BOOL:= FALSE;
	bEnCheck : REFERENCE TO BOOL;
END_VAR
VAR
	fbEnclosureSensorFilter: fbBinaryFilter;
	bPartInFixture: BOOL;
	bPartWelded: BOOL;
	iCtr_SensorWorkVerification: INT;	// Value reset at every part pull up from fixture
END_VAR

// Filtrowanie sygnału z czujnika obudowy
fbEnclosureSensorFilter(IN := (stInOuts.bEnclosureSensor XOR bEnclosureSensorInvert) OR NOT bEnCheck, tON := tSensorFilterTime, tOFF := tSensorFilterTime/2);
bPartInFixture S= fbEnclosureSensorFilter.RTrig;

IF fbEnclosureSensorFilter.FTrig THEN	// Wyjęcie części z kowadła
	IF bEnCheck AND bPartInFixture AND NOT bPartWelded THEN
		nQErrorId := nStFix_S17EnclosureWelding_ErrorCodes.PartsNotWelded;
		iWorkStep := 90;
	ELSE
		bPartInFixture := bPartWelded := FALSE;
	END_IF
	iCtr_SensorWorkVerification := 0;	
END_IF

